LIN {X 0,Y 488.725,Z 497.921,A -85,B 0,C 180,E1 -6513.485,E2 -6513.485} C_VEL
LIN {X 0,Y 488.681,Z 497.925,A -85,B 0,C 180,E1 -6516.357,E2 -6516.357} C_VEL
LIN {X 0,Y 488.74,Z 497.918,A -85,B 0,C 180,E1 -6519.25,E2 -6519.25} C_VEL
LIN {X 0,Y 488.724,Z 497.922,A -85,B 0,C 180,E1 -6522.522,E2 -6522.522} C_VEL
LIN {X 0,Y 488.717,Z 498.007,A -85,B 0,C 180,E1 -6523.954,E2 -6523.954} C_VEL
LIN {X 0,Y 490.803,Z 507.385,A -85,B 0,C 180,E1 -6526.91,E2 -6526.91} C_VEL
LIN {X 0,Y 492.374,Z 514.903,A -85,B 0,C 180,E1 -6529.157,E2 -6529.157} C_VEL
LIN {X 0,Y 492.613,Z 519.318,A -85,B 0,C 180,E1 -6530.39,E2 -6530.39} C_VEL
LIN {X 0,Y 492.156,Z 529.697,A -85,B 0,C 180,E1 -6533.149,E2 -6533.149} C_VEL
LIN {X 0,Y 491.624,Z 540.769,A -85,B 0,C 180,E1 -6536.01,E2 -6536.01} C_VEL
LIN {X 0,Y 491.178,Z 552.868,A -85,B 0,C 180,E1 -6538.997,E2 -6538.997} C_VEL
LIN {X 0,Y 490.723,Z 566.378,A -85,B 0,C 180,E1 -6542.262,E2 -6542.262} C_VEL
LIN {X 0,Y 490.185,Z 577.141,A -85,B 0,C 180,E1 -6544.944,E2 -6544.944} C_VEL
LIN {X 0,Y 496.327,Z 599.12,A -85,B 0,C 180,E1 -6545.676,E2 -6545.676} C_VEL
LIN {X 0,Y 496.647,Z 602.392,A -85,B 0,C 180,E1 -6545.773,E2 -6545.773} C_VEL
LIN {X 0,Y 496.101,Z 618.413,A -85,B 0,C 180,E1 -6546.242,E2 -6546.242} C_VEL
LIN {X 0,Y 495.355,Z 634.974,A -85,B 0,C 180,E1 -6546.898,E2 -6546.898} C_VEL
LIN {X 0,Y 494.605,Z 650.253,A -85,B 0,C 180,E1 -6547.677,E2 -6547.677} C_VEL
LIN {X 0,Y 493.629,Z 665.049,A -85,B 0,C 180,E1 -6548.604,E2 -6548.604} C_VEL
LIN {X 0,Y 492.776,Z 678.915,A -85,B 0,C 180,E1 -6549.658,E2 -6549.658} C_VEL
LIN {X 0,Y 491.84,Z 691.852,A -85,B 0,C 180,E1 -6550.814,E2 -6550.814} C_VEL
LIN {X 0,Y 491.019,Z 703.949,A -85,B 0,C 180,E1 -6552.079,E2 -6552.079} C_VEL
LIN {X 0,Y 490.241,Z 715.847,A -85,B 0,C 180,E1 -6553.548,E2 -6553.548} C_VEL
LIN {X 0,Y 489.589,Z 726.058,A -85,B 0,C 180,E1 -6555.027,E2 -6555.027} C_VEL
LIN {X 0,Y 488.981,Z 735.94,A -85,B 0,C 180,E1 -6556.706,E2 -6556.706} C_VEL
LIN {X 0,Y 488.619,Z 744.242,A -85,B 0,C 180,E1 -6558.384,E2 -6558.384} C_VEL
LIN {X 0,Y 488.232,Z 751.104,A -85,B 0,C 180,E1 -6560.054,E2 -6560.054} C_VEL
LIN {X 0,Y 488.096,Z 756.719,A -85,B 0,C 180,E1 -6561.722,E2 -6561.722} C_VEL
LIN {X 0,Y 488.006,Z 761.657,A -85,B 0,C 180,E1 -6563.563,E2 -6563.563} C_VEL
LIN {X 0,Y 487.908,Z 764.636,A -85,B 0,C 180,E1 -6565.043,E2 -6565.043} C_VEL
LIN {X 0,Y 487.944,Z 767.091,A -85,B 0,C 180,E1 -6566.698,E2 -6566.698} C_VEL
LIN {X 0,Y 487.884,Z 768.479,A -85,B 0,C 180,E1 -6568.35,E2 -6568.35} C_VEL
LIN {X 0,Y 487.814,Z 769,A -85,B 0,C 180,E1 -6570.001,E2 -6570.001} C_VEL
LIN {X 0,Y 487.884,Z 768.478,A -85,B 0,C 180,E1 -6571.652,E2 -6571.652} C_VEL
LIN {X 0,Y 487.944,Z 767.088,A -85,B 0,C 180,E1 -6573.304,E2 -6573.304} C_VEL
LIN {X 0,Y 487.909,Z 764.633,A -85,B 0,C 180,E1 -6574.959,E2 -6574.959} C_VEL
LIN {X 0,Y 488.028,Z 761.249,A -85,B 0,C 180,E1 -6576.616,E2 -6576.616} C_VEL
LIN {X 0,Y 488.124,Z 755.465,A -85,B 0,C 180,E1 -6578.696,E2 -6578.696} C_VEL
LIN {X 0,Y 488.432,Z 747.853,A -85,B 0,C 180,E1 -6580.782,E2 -6580.782} C_VEL
LIN {X 0,Y 488.824,Z 739.251,A -85,B 0,C 180,E1 -6582.666,E2 -6582.666} C_VEL
LIN {X 0,Y 489.347,Z 729.973,A -85,B 0,C 180,E1 -6584.345,E2 -6584.345} C_VEL
LIN {X 0,Y 489.928,Z 720.416,A -85,B 0,C 180,E1 -6585.817,E2 -6585.817} C_VEL
LIN {X 0,Y 490.659,Z 709.277,A -85,B 0,C 180,E1 -6587.291,E2 -6587.291} C_VEL
LIN {X 0,Y 491.496,Z 697.133,A -85,B 0,C 180,E1 -6588.66,E2 -6588.66} C_VEL
LIN {X 0,Y 492.417,Z 683.772,A -85,B 0,C 180,E1 -6589.932,E2 -6589.932} C_VEL
LIN {X 0,Y 493.382,Z 669.408,A -85,B 0,C 180,E1 -6591.081,E2 -6591.081} C_VEL
LIN {X 0,Y 494.346,Z 654.423,A -85,B 0,C 180,E1 -6592.075,E2 -6592.075} C_VEL
LIN {X 0,Y 495.141,Z 640.233,A -85,B 0,C 180,E1 -6592.854,E2 -6592.854} C_VEL
LIN {X 0,Y 495.855,Z 625.368,A -85,B 0,C 180,E1 -6593.504,E2 -6593.504} C_VEL
LIN {X 0,Y 496.412,Z 608.983,A -85,B 0,C 180,E1 -6594.055,E2 -6594.055} C_VEL
LIN {X 0,Y 496.555,Z 600.107,A -85,B 0,C 180,E1 -6594.288,E2 -6594.288} C_VEL
LIN {X 0,Y 490.963,Z 580.048,A -85,B 0,C 180,E1 -6594.966,E2 -6594.966} C_VEL
LIN {X 0,Y 490.197,Z 577.068,A -85,B 0,C 180,E1 -6595.073,E2 -6595.073} C_VEL
LIN {X 0,Y 490.764,Z 564.422,A -85,B 0,C 180,E1 -6598.202,E2 -6598.202} C_VEL
LIN {X 0,Y 491.068,Z 550.504,A -85,B 0,C 180,E1 -6601.252,E2 -6601.252} C_VEL
LIN {X 0,Y 491.235,Z 537.358,A -85,B 0,C 180,E1 -6604.163,E2 -6604.163} C_VEL
LIN {X 0,Y 491.399,Z 525.732,A -85,B 0,C 180,E1 -6606.783,E2 -6606.783} C_VEL
LIN {X 0,Y 491.485,Z 513.366,A -85,B 0,C 180,E1 -6609.707,E2 -6609.707} C_VEL
LIN {X 0,Y 490.808,Z 508.373,A -85,B 0,C 180,E1 -6611,E2 -6611} C_VEL
LIN {X 0,Y 489.018,Z 499.36,A -85,B 0,C 180,E1 -6613.618,E2 -6613.618} C_VEL
LIN {X 0,Y 488.71,Z 497.924,A -85,B 0,C 180,E1 -6614.132,E2 -6614.132} C_VEL
LIN {X 0,Y 488.716,Z 497.923,A -85,B 0,C 180,E1 -6617.173,E2 -6617.173} C_VEL
LIN {X 0,Y 488.734,Z 497.919,A -85,B 0,C 180,E1 -6619.677,E2 -6619.677} C_VEL
LIN {X 0,Y 488.683,Z 497.927,A -85,B 0,C 180,E1 -6622.842,E2 -6622.842} C_VEL
LIN {X 0,Y 488.735,Z 497.92,A -85,B 0,C 180,E1 -6625.888,E2 -6625.888} C_VEL
LIN {X 0,Y 488.694,Z 497.925,A -85,B 0,C 180,E1 -6628.821,E2 -6628.821} C_VEL
LIN {X 0,Y 488.747,Z 497.919,A -85,B 0,C 180,E1 -6631.672,E2 -6631.672} C_VEL
LIN {X 0,Y 488.749,Z 497.919,A -85,B 0,C 180,E1 -6634.445,E2 -6634.445} C_VEL
LIN {X 0,Y 488.776,Z 498.087,A -85,B 0,C 180,E1 -6635.425,E2 -6635.425} C_VEL
LIN {X 0,Y 491.571,Z 505.225,A -85,B 0,C 180,E1 -6635.733,E2 -6635.733} C_VEL
LIN {X 0,Y 495.968,Z 516.083,A -85,B 0,C 180,E1 -6636.261,E2 -6636.261} C_VEL
LIN {X 0,Y 495.474,Z 531.577,A -85,B 0,C 180,E1 -6636.821,E2 -6636.821} C_VEL
LIN {X 0,Y 494.777,Z 546.893,A -85,B 0,C 180,E1 -6637.528,E2 -6637.528} C_VEL
LIN {X 0,Y 493.954,Z 562.027,A -85,B 0,C 180,E1 -6638.399,E2 -6638.399} C_VEL
LIN {X 0,Y 493.106,Z 576.875,A -85,B 0,C 180,E1 -6639.454,E2 -6639.454} C_VEL
LIN {X 0,Y 492.154,Z 590.761,A -85,B 0,C 180,E1 -6640.643,E2 -6640.643} C_VEL
LIN {X 0,Y 491.351,Z 602.834,A -85,B 0,C 180,E1 -6641.875,E2 -6641.875} C_VEL
LIN {X 0,Y 490.498,Z 615.066,A -85,B 0,C 180,E1 -6643.348,E2 -6643.348} C_VEL
LIN {X 0,Y 489.846,Z 625.403,A -85,B 0,C 180,E1 -6644.821,E2 -6644.821} C_VEL
LIN {X 0,Y 489.215,Z 634.165,A -85,B 0,C 180,E1 -6646.289,E2 -6646.289} C_VEL
LIN {X 0,Y 488.786,Z 643.123,A -85,B 0,C 180,E1 -6648.079,E2 -6648.079} C_VEL
LIN {X 0,Y 488.353,Z 649.619,A -85,B 0,C 180,E1 -6649.637,E2 -6649.637} C_VEL
LIN {X 0,Y 488.136,Z 655.35,A -85,B 0,C 180,E1 -6651.305,E2 -6651.305} C_VEL
LIN {X 0,Y 488.047,Z 660.122,A -85,B 0,C 180,E1 -6652.97,E2 -6652.97} C_VEL
LIN {X 0,Y 487.91,Z 664.571,A -85,B 0,C 180,E1 -6655.042,E2 -6655.042} C_VEL
LIN {X 0,Y 487.947,Z 667.016,A -85,B 0,C 180,E1 -6656.698,E2 -6656.698} C_VEL
LIN {X 0,Y 487.884,Z 668.488,A -85,B 0,C 180,E1 -6658.349,E2 -6658.349} C_VEL
LIN {X 0,Y 487.817,Z 668.997,A -85,B 0,C 180,E1 -6660,E2 -6660} C_VEL
LIN {X 0,Y 487.884,Z 668.527,A -85,B 0,C 180,E1 -6661.651,E2 -6661.651} C_VEL
LIN {X 0,Y 487.948,Z 667.112,A -85,B 0,C 180,E1 -6663.303,E2 -6663.303} C_VEL
LIN {X 0,Y 487.91,Z 664.728,A -85,B 0,C 180,E1 -6664.958,E2 -6664.958} C_VEL
LIN {X 0,Y 488.032,Z 661.294,A -85,B 0,C 180,E1 -6666.633,E2 -6666.633} C_VEL
LIN {X 0,Y 488.096,Z 656.884,A -85,B 0,C 180,E1 -6668.279,E2 -6668.279} C_VEL
LIN {X 0,Y 488.339,Z 649.846,A -85,B 0,C 180,E1 -6670.364,E2 -6670.364} C_VEL
LIN {X 0,Y 488.751,Z 642.59,A -85,B 0,C 180,E1 -6672.093,E2 -6672.093} C_VEL
LIN {X 0,Y 489.171,Z 634.413,A -85,B 0,C 180,E1 -6673.713,E2 -6673.713} C_VEL
LIN {X 0,Y 489.861,Z 624.292,A -85,B 0,C 180,E1 -6675.392,E2 -6675.392} C_VEL
LIN {X 0,Y 490.52,Z 613.752,A -85,B 0,C 180,E1 -6676.866,E2 -6676.866} C_VEL
LIN {X 0,Y 491.346,Z 601.265,A -85,B 0,C 180,E1 -6678.342,E2 -6678.342} C_VEL
LIN {X 0,Y 492.299,Z 588.147,A -85,B 0,C 180,E1 -6679.646,E2 -6679.646} C_VEL
LIN {X 0,Y 493.142,Z 574.876,A -85,B 0,C 180,E1 -6680.764,E2 -6680.764} C_VEL
LIN {X 0,Y 494.088,Z 560.086,A -85,B 0,C 180,E1 -6681.8,E2 -6681.8} C_VEL
LIN {X 0,Y 494.967,Z 543.931,A -85,B 0,C 180,E1 -6682.722,E2 -6682.722} C_VEL
LIN {X 0,Y 495.702,Z 527.836,A -85,B 0,C 180,E1 -6683.442,E2 -6683.442} C_VEL
LIN {X 0,Y 495.996,Z 515.787,A -85,B 0,C 180,E1 -6683.882,E2 -6683.882} C_VEL
LIN {X 0,Y 488.905,Z 498.693,A -85,B 0,C 180,E1 -6684.723,E2 -6684.723} C_VEL
LIN {X 0,Y 488.751,Z 497.919,A -85,B 0,C 180,E1 -6684.776,E2 -6684.776} C_VEL
LIN {X 0,Y 488.75,Z 497.919,A -85,B 0,C 180,E1 -6687.397,E2 -6687.397} C_VEL
LIN {X 0,Y 488.714,Z 497.924,A -85,B 0,C 180,E1 -6690.363,E2 -6690.363} C_VEL
LIN {X 0,Y 488.74,Z 497.92,A -85,B 0,C 180,E1 -6693.484,E2 -6693.484} C_VEL
LIN {X 0,Y 488.693,Z 497.925,A -85,B 0,C 180,E1 -6696.356,E2 -6696.356} C_VEL
LIN {X 0,Y 488.706,Z 497.923,A -85,B 0,C 180,E1 -6699.254,E2 -6699.254} C_VEL
LIN {X 0,Y 488.711,Z 497.924,A -85,B 0,C 180,E1 -6701.6,E2 -6701.6} C_VEL
LIN {X 0,Y 488.706,Z 497.924,A -85,B 0,C 180,E1 -6704.803,E2 -6704.803} C_VEL
LIN {X 0,Y 488.697,Z 497.927,A -85,B 0,C 180,E1 -6707.475,E2 -6707.475} C_VEL
LIN {X 0,Y 488.738,Z 497.918,A -85,B 0,C 180,E1 -6709.677,E2 -6709.677} C_VEL
LIN {X 0,Y 488.685,Z 497.926,A -85,B 0,C 180,E1 -6712.841,E2 -6712.841} C_VEL
LIN {X 0,Y 488.72,Z 497.921,A -85,B 0,C 180,E1 -6715.293,E2 -6715.293} C_VEL
LIN {X 0,Y 488.045,Z 498.009,A -85,B 0,C 180,E1 -6715.981,E2 -6715.981} C_VEL
LIN {X 0,Y 485.167,Z 498.367,A -85,B 0,C 180,E1 -6717.098,E2 -6717.098} C_VEL
LIN {X 0,Y 482.742,Z 498.669,A -85,B 0,C 180,E1 -6717.998,E2 -6717.998} C_VEL
LIN {X 0,Y 481.713,Z 498.799,A -85,B 0,C 180,E1 -6718.694,E2 -6718.694} C_VEL
LIN {X 0,Y 481.635,Z 498.805,A -85,B 0,C 180,E1 -6718.93,E2 -6718.93} C_VEL
LIN {X 0,Y 481.705,Z 498.797,A -85,B 0,C 180,E1 -6721.218,E2 -6721.218} C_VEL
LIN {X 0,Y 481.721,Z 498.795,A -85,B 0,C 180,E1 -6724.043,E2 -6724.043} C_VEL
LIN {X 0,Y 481.809,Z 498.814,A -85,B 0,C 180,E1 -6725.09,E2 -6725.09} C_VEL
LIN {X 0,Y 481.825,Z 503.568,A -85,B 0,C 180,E1 -6727.713,E2 -6727.713} C_VEL
LIN {X 0,Y 481.792,Z 508.356,A -85,B 0,C 180,E1 -6730.396,E2 -6730.396} C_VEL
LIN {X 0,Y 481.714,Z 512.928,A -85,B 0,C 180,E1 -6733.034,E2 -6733.034} C_VEL
LIN {X 0,Y 481.656,Z 517.34,A -85,B 0,C 180,E1 -6735.637,E2 -6735.637} C_VEL
LIN {X 0,Y 481.655,Z 521.628,A -85,B 0,C 180,E1 -6738.212,E2 -6738.212} C_VEL
LIN {X 0,Y 481.521,Z 523.894,A -85,B 0,C 180,E1 -6739.585,E2 -6739.585} C_VEL
LIN {X 0,Y 483.194,Z 528.751,A -85,B 0,C 180,E1 -6739.766,E2 -6739.766} C_VEL
LIN {X 0,Y 487.776,Z 541.51,A -85,B 0,C 180,E1 -6740.284,E2 -6740.284} C_VEL
LIN {X 0,Y 490.122,Z 549.845,A -85,B 0,C 180,E1 -6740.638,E2 -6740.638} C_VEL
LIN {X 0,Y 489.482,Z 566.262,A -85,B 0,C 180,E1 -6741.187,E2 -6741.187} C_VEL
LIN {X 0,Y 488.681,Z 581.972,A -85,B 0,C 180,E1 -6741.887,E2 -6741.887} C_VEL
LIN {X 0,Y 487.896,Z 595.778,A -85,B 0,C 180,E1 -6742.654,E2 -6742.654} C_VEL
LIN {X 0,Y 486.995,Z 609.618,A -85,B 0,C 180,E1 -6743.578,E2 -6743.578} C_VEL
LIN {X 0,Y 485.954,Z 623.681,A -85,B 0,C 180,E1 -6744.709,E2 -6744.709} C_VEL
LIN {X 0,Y 484.982,Z 636.591,A -85,B 0,C 180,E1 -6745.948,E2 -6745.948} C_VEL
LIN {X 0,Y 484.042,Z 648.549,A -85,B 0,C 180,E1 -6747.294,E2 -6747.294} C_VEL
LIN {X 0,Y 483.242,Z 659.576,A -85,B 0,C 180,E1 -6748.749,E2 -6748.749} C_VEL
LIN {X 0,Y 482.389,Z 670.303,A -85,B 0,C 180,E1 -6750.416,E2 -6750.416} C_VEL
LIN {X 0,Y 481.88,Z 679.281,A -85,B 0,C 180,E1 -6752.089,E2 -6752.089} C_VEL
LIN {X 0,Y 481.43,Z 686.808,A -85,B 0,C 180,E1 -6753.766,E2 -6753.766} C_VEL
LIN {X 0,Y 481.158,Z 693.144,A -85,B 0,C 180,E1 -6755.447,E2 -6755.447} C_VEL
LIN {X 0,Y 480.967,Z 699.432,A -85,B 0,C 180,E1 -6757.556,E2 -6757.556} C_VEL
LIN {X 0,Y 480.779,Z 703.245,A -85,B 0,C 180,E1 -6759.252,E2 -6759.252} C_VEL
LIN {X 0,Y 480.778,Z 706.068,A -85,B 0,C 180,E1 -6760.954,E2 -6760.954} C_VEL
LIN {X 0,Y 480.792,Z 707.203,A -85,B 0,C 180,E1 -6761.808,E2 -6761.808} C_VEL
LIN {X 0,Y 480.678,Z 708.608,A -85,B 0,C 180,E1 -6763.528,E2 -6763.528} C_VEL
LIN {X 0,Y 480.686,Z 708.958,A -85,B 0,C 180,E1 -6765.257,E2 -6765.257} C_VEL
LIN {X 0,Y 480.664,Z 708.286,A -85,B 0,C 180,E1 -6767.002,E2 -6767.002} C_VEL
LIN {X 0,Y 480.708,Z 707.376,A -85,B 0,C 180,E1 -6768.137,E2 -6768.137} C_VEL
LIN {X 0,Y 480.706,Z 705.387,A -85,B 0,C 180,E1 -6769.648,E2 -6769.648} C_VEL
LIN {X 0,Y 480.85,Z 702.058,A -85,B 0,C 180,E1 -6771.431,E2 -6771.431} C_VEL
LIN {X 0,Y 480.972,Z 697.519,A -85,B 0,C 180,E1 -6773.235,E2 -6773.235} C_VEL
LIN {X 0,Y 481.173,Z 693.316,A -85,B 0,C 180,E1 -6774.598,E2 -6774.598} C_VEL
LIN {X 0,Y 481.49,Z 686.376,A -85,B 0,C 180,E1 -6776.434,E2 -6776.434} C_VEL
LIN {X 0,Y 481.874,Z 679.039,A -85,B 0,C 180,E1 -6778.056,E2 -6778.056} C_VEL
LIN {X 0,Y 482.471,Z 670.265,A -85,B 0,C 180,E1 -6779.686,E2 -6779.686} C_VEL
LIN {X 0,Y 483.229,Z 659.526,A -85,B 0,C 180,E1 -6781.359,E2 -6781.359} C_VEL
LIN {X 0,Y 484.128,Z 648.196,A -85,B 0,C 180,E1 -6782.847,E2 -6782.847} C_VEL
LIN {X 0,Y 485.03,Z 636.036,A -85,B 0,C 180,E1 -6784.209,E2 -6784.209} C_VEL
LIN {X 0,Y 485.99,Z 623.103,A -85,B 0,C 180,E1 -6785.441,E2 -6785.441} C_VEL
LIN {X 0,Y 486.981,Z 609.495,A -85,B 0,C 180,E1 -6786.533,E2 -6786.533} C_VEL
LIN {X 0,Y 488.011,Z 593.857,A -85,B 0,C 180,E1 -6787.565,E2 -6787.565} C_VEL
LIN {X 0,Y 488.853,Z 578.577,A -85,B 0,C 180,E1 -6788.378,E2 -6788.378} C_VEL
LIN {X 0,Y 489.58,Z 563.019,A -85,B 0,C 180,E1 -6789.03,E2 -6789.03} C_VEL
LIN {X 0,Y 490.006,Z 549.235,A -85,B 0,C 180,E1 -6789.482,E2 -6789.482} C_VEL
LIN {X 0,Y 485.726,Z 535.434,A -85,B 0,C 180,E1 -6790.056,E2 -6790.056} C_VEL
LIN {X 0,Y 481.567,Z 524.772,A -85,B 0,C 180,E1 -6790.484,E2 -6790.484} C_VEL
LIN {X 0,Y 481.449,Z 524.174,A -85,B 0,C 180,E1 -6790.505,E2 -6790.505} C_VEL
LIN {X 0,Y 481.573,Z 519.519,A -85,B 0,C 180,E1 -6793.305,E2 -6793.305} C_VEL
LIN {X 0,Y 481.703,Z 515.606,A -85,B 0,C 180,E1 -6795.633,E2 -6795.633} C_VEL
LIN {X 0,Y 481.784,Z 509.992,A -85,B 0,C 180,E1 -6798.971,E2 -6798.971} C_VEL
LIN {X 0,Y 481.814,Z 504.644,A -85,B 0,C 180,E1 -6801.966,E2 -6801.966} C_VEL
LIN {X 0,Y 481.871,Z 500.416,A -85,B 0,C 180,E1 -6804.31,E2 -6804.31} C_VEL
LIN {X 0,Y 481.719,Z 498.796,A -85,B 0,C 180,E1 -6805.25,E2 -6805.25} C_VEL
LIN {X 0,Y 481.641,Z 498.808,A -85,B 0,C 180,E1 -6808.311,E2 -6808.311} C_VEL
LIN {X 0,Y 481.699,Z 498.797,A -85,B 0,C 180,E1 -6811.218,E2 -6811.218} C_VEL
LIN {X 0,Y 481.699,Z 498.797,A -85,B 0,C 180,E1 -6814.042,E2 -6814.042} C_VEL
LIN {X 0,Y 481.665,Z 498.799,A -85,B 0,C 180,E1 -6816.811,E2 -6816.811} C_VEL
LIN {X 0,Y 481.689,Z 498.798,A -85,B 0,C 180,E1 -6819.502,E2 -6819.502} C_VEL
LIN {X 0,Y 481.698,Z 498.797,A -85,B 0,C 180,E1 -6822.158,E2 -6822.158} C_VEL
LIN {X 0,Y 481.732,Z 498.792,A -85,B 0,C 180,E1 -6824.775,E2 -6824.775} C_VEL
LIN {X 0,Y 481.785,Z 498.787,A -85,B 0,C 180,E1 -6828.216,E2 -6828.216} C_VEL
LIN {X 0,Y 481.754,Z 498.785,A -85,B 0,C 180,E1 -6831.611,E2 -6831.611} C_VEL
LIN {X 0,Y 481.822,Z 498.78,A -85,B 0,C 180,E1 -6834.139,E2 -6834.139} C_VEL
LIN {X 0,Y 481.92,Z 498.768,A -85,B 0,C 180,E1 -6837.492,E2 -6837.492} C_VEL
LIN {X 0,Y 481.929,Z 498.767,A -85,B 0,C 180,E1 -6840,E2 -6840} C_VEL
LIN {X 0,Y 481.92,Z 498.766,A -85,B 0,C 180,E1 -6842.507,E2 -6842.507} C_VEL
LIN {X 0,Y 481.806,Z 498.777,A -85,B 0,C 180,E1 -6845.86,E2 -6845.86} C_VEL
LIN {X 0,Y 481.753,Z 498.786,A -85,B 0,C 180,E1 -6848.388,E2 -6848.388} C_VEL
LIN {X 0,Y 481.784,Z 498.781,A -85,B 0,C 180,E1 -6851.784,E2 -6851.784} C_VEL
LIN {X 0,Y 481.731,Z 498.79,A -85,B 0,C 180,E1 -6855.224,E2 -6855.224} C_VEL
LIN {X 0,Y 481.701,Z 498.782,A -85,B 0,C 180,E1 -6858.722,E2 -6858.722} C_VEL
LIN {X 0,Y 481.661,Z 498.801,A -85,B 0,C 180,E1 -6861.394,E2 -6861.394} C_VEL
LIN {X 0,Y 481.671,Z 498.78,A -85,B 0,C 180,E1 -6864.113,E2 -6864.113} C_VEL
LIN {X 0,Y 481.741,Z 498.79,A -85,B 0,C 180,E1 -6867.141,E2 -6867.141} C_VEL
LIN {X 0,Y 481.677,Z 498.798,A -85,B 0,C 180,E1 -6869.741,E2 -6869.741} C_VEL
LIN {X 0,Y 481.663,Z 498.8,A -85,B 0,C 180,E1 -6872.674,E2 -6872.674} C_VEL
LIN {X 0,Y 481.634,Z 498.803,A -85,B 0,C 180,E1 -6875.709,E2 -6875.709} C_VEL
LIN {X 0,Y 481.713,Z 498.793,A -85,B 0,C 180,E1 -6879.356,E2 -6879.356} C_VEL
LIN {X 0,Y 481.666,Z 498.801,A -85,B 0,C 180,E1 -6882.158,E2 -6882.158} C_VEL
LIN {X 0,Y 481.684,Z 498.854,A -85,B 0,C 180,E1 -6883.51,E2 -6883.51} C_VEL
LIN {X 0,Y 483.777,Z 508.43,A -85,B 0,C 180,E1 -6886.582,E2 -6886.582} C_VEL
LIN {X 0,Y 485.385,Z 515.824,A -85,B 0,C 180,E1 -6888.843,E2 -6888.843} C_VEL
LIN {X 0,Y 485.754,Z 520.091,A -85,B 0,C 180,E1 -6890.068,E2 -6890.068} C_VEL
LIN {X 0,Y 485.357,Z 529.232,A -85,B 0,C 180,E1 -6892.545,E2 -6892.545} C_VEL
LIN {X 0,Y 484.909,Z 538.824,A -85,B 0,C 180,E1 -6895.077,E2 -6895.077} C_VEL
LIN {X 0,Y 484.371,Z 550.439,A -85,B 0,C 180,E1 -6898.023,E2 -6898.023} C_VEL
LIN {X 0,Y 483.892,Z 562.462,A -85,B 0,C 180,E1 -6900.988,E2 -6900.988} C_VEL
LIN {X 0,Y 483.456,Z 573.592,A -85,B 0,C 180,E1 -6903.682,E2 -6903.682} C_VEL
LIN {X 0,Y 483.296,Z 577.121,A -85,B 0,C 180,E1 -6904.557,E2 -6904.557} C_VEL
LIN {X 0,Y 489.432,Z 599.121,A -85,B 0,C 180,E1 -6905.311,E2 -6905.311} C_VEL
LIN {X 0,Y 490.174,Z 602.392,A -85,B 0,C 180,E1 -6905.432,E2 -6905.432} C_VEL
LIN {X 0,Y 489.584,Z 618.966,A -85,B 0,C 180,E1 -6905.926,E2 -6905.926} C_VEL
LIN {X 0,Y 488.79,Z 635.537,A -85,B 0,C 180,E1 -6906.598,E2 -6906.598} C_VEL
LIN {X 0,Y 487.97,Z 650.948,A -85,B 0,C 180,E1 -6907.401,E2 -6907.401} C_VEL
LIN {X 0,Y 486.966,Z 665.051,A -85,B 0,C 180,E1 -6908.296,E2 -6908.296} C_VEL
LIN {X 0,Y 486.072,Z 678.913,A -85,B 0,C 180,E1 -6909.365,E2 -6909.365} C_VEL
LIN {X 0,Y 484.978,Z 692.92,A -85,B 0,C 180,E1 -6910.642,E2 -6910.642} C_VEL
LIN {X 0,Y 484.036,Z 705.732,A -85,B 0,C 180,E1 -6912.03,E2 -6912.03} C_VEL
LIN {X 0,Y 483.198,Z 717.701,A -85,B 0,C 180,E1 -6913.56,E2 -6913.56} C_VEL
LIN {X 0,Y 482.561,Z 727.411,A -85,B 0,C 180,E1 -6915.019,E2 -6915.019} C_VEL
LIN {X 0,Y 481.902,Z 737.055,A -85,B 0,C 180,E1 -6916.722,E2 -6916.722} C_VEL
LIN {X 0,Y 481.612,Z 744.243,A -85,B 0,C 180,E1 -6918.213,E2 -6918.213} C_VEL
LIN {X 0,Y 481.185,Z 751.103,A -85,B 0,C 180,E1 -6919.907,E2 -6919.907} C_VEL
LIN {X 0,Y 481.023,Z 756.719,A -85,B 0,C 180,E1 -6921.6,E2 -6921.6} C_VEL
LIN {X 0,Y 480.917,Z 761.897,A -85,B 0,C 180,E1 -6923.58,E2 -6923.58} C_VEL
LIN {X 0,Y 480.834,Z 764.636,A -85,B 0,C 180,E1 -6924.97,E2 -6924.97} C_VEL
LIN {X 0,Y 480.849,Z 767.091,A -85,B 0,C 180,E1 -6926.649,E2 -6926.649} C_VEL
LIN {X 0,Y 480.785,Z 768.479,A -85,B 0,C 180,E1 -6928.326,E2 -6928.326} C_VEL
LIN {X 0,Y 480.738,Z 769,A -85,B 0,C 180,E1 -6930.001,E2 -6930.001} C_VEL
LIN {X 0,Y 480.785,Z 768.478,A -85,B 0,C 180,E1 -6931.676,E2 -6931.676} C_VEL
LIN {X 0,Y 480.85,Z 767.088,A -85,B 0,C 180,E1 -6933.352,E2 -6933.352} C_VEL
LIN {X 0,Y 480.835,Z 764.633,A -85,B 0,C 180,E1 -6935.032,E2 -6935.032} C_VEL
LIN {X 0,Y 480.951,Z 761.249,A -85,B 0,C 180,E1 -6936.714,E2 -6936.714} C_VEL
LIN {X 0,Y 481.058,Z 755.465,A -85,B 0,C 180,E1 -6938.825,E2 -6938.825} C_VEL
LIN {X 0,Y 481.399,Z 747.853,A -85,B 0,C 180,E1 -6940.941,E2 -6940.941} C_VEL
LIN {X 0,Y 481.822,Z 739.252,A -85,B 0,C 180,E1 -6942.853,E2 -6942.853} C_VEL
LIN {X 0,Y 482.366,Z 729.973,A -85,B 0,C 180,E1 -6944.557,E2 -6944.557} C_VEL
LIN {X 0,Y 482.998,Z 720.416,A -85,B 0,C 180,E1 -6946.05,E2 -6946.05} C_VEL
LIN {X 0,Y 483.784,Z 709.277,A -85,B 0,C 180,E1 -6947.545,E2 -6947.545} C_VEL
LIN {X 0,Y 484.702,Z 697.132,A -85,B 0,C 180,E1 -6948.932,E2 -6948.932} C_VEL
LIN {X 0,Y 485.686,Z 683.868,A -85,B 0,C 180,E1 -6950.211,E2 -6950.211} C_VEL
LIN {X 0,Y 486.61,Z 670.833,A -85,B 0,C 180,E1 -6951.278,E2 -6951.278} C_VEL
LIN {X 0,Y 487.614,Z 656.231,A -85,B 0,C 180,E1 -6952.282,E2 -6952.282} C_VEL
LIN {X 0,Y 488.479,Z 642.089,A -85,B 0,C 180,E1 -6953.083,E2 -6953.083} C_VEL
LIN {X 0,Y 489.274,Z 626.871,A -85,B 0,C 180,E1 -6953.775,E2 -6953.775} C_VEL
LIN {X 0,Y 489.863,Z 611.154,A -85,B 0,C 180,E1 -6954.33,E2 -6954.33} C_VEL
LIN {X 0,Y 490.106,Z 601.692,A -85,B 0,C 180,E1 -6954.589,E2 -6954.589} C_VEL
LIN {X 0,Y 485.5,Z 584.865,A -85,B 0,C 180,E1 -6955.189,E2 -6955.189} C_VEL
LIN {X 0,Y 483.293,Z 577.11,A -85,B 0,C 180,E1 -6955.446,E2 -6955.446} C_VEL
LIN {X 0,Y 483.562,Z 569.778,A -85,B 0,C 180,E1 -6957.178,E2 -6957.178} C_VEL
LIN {X 0,Y 483.873,Z 556.679,A -85,B 0,C 180,E1 -6960.073,E2 -6960.073} C_VEL
LIN {X 0,Y 484.154,Z 543.502,A -85,B 0,C 180,E1 -6963.02,E2 -6963.02} C_VEL
LIN {X 0,Y 484.358,Z 530.237,A -85,B 0,C 180,E1 -6966.041,E2 -6966.041} C_VEL
LIN {X 0,Y 484.561,Z 517.337,A -85,B 0,C 180,E1 -6969.118,E2 -6969.118} C_VEL
LIN {X 0,Y 484.476,Z 513.014,A -85,B 0,C 180,E1 -6970.211,E2 -6970.211} C_VEL
LIN {X 0,Y 482.812,Z 504.327,A -85,B 0,C 180,E1 -6972.686,E2 -6972.686} C_VEL
LIN {X 0,Y 481.674,Z 498.801,A -85,B 0,C 180,E1 -6974.529,E2 -6974.529} C_VEL
LIN {X 0,Y 481.655,Z 498.801,A -85,B 0,C 180,E1 -6977.841,E2 -6977.841} C_VEL
LIN {X 0,Y 481.682,Z 498.8,A -85,B 0,C 180,E1 -6980.652,E2 -6980.652} C_VEL
LIN {X 0,Y 481.631,Z 498.804,A -85,B 0,C 180,E1 -6983.376,E2 -6983.376} C_VEL
LIN {X 0,Y 481.711,Z 498.797,A -85,B 0,C 180,E1 -6986.331,E2 -6986.331} C_VEL
LIN {X 0,Y 481.652,Z 498.801,A -85,B 0,C 180,E1 -6989.418,E2 -6989.418} C_VEL
LIN {X 0,Y 481.702,Z 498.798,A -85,B 0,C 180,E1 -6992.169,E2 -6992.169} C_VEL
LIN {X 0,Y 481.709,Z 498.795,A -85,B 0,C 180,E1 -6995.072,E2 -6995.072} C_VEL
LIN {X 0,Y 483.396,Z 503.34,A -85,B 0,C 180,E1 -6995.264,E2 -6995.264} C_VEL
LIN {X 0,Y 489.358,Z 518.074,A -85,B 0,C 180,E1 -6996,E2 -6996} C_VEL
LIN {X 0,Y 488.788,Z 534.305,A -85,B 0,C 180,E1 -6996.612,E2 -6996.612} C_VEL
LIN {X 0,Y 488.059,Z 549.801,A -85,B 0,C 180,E1 -6997.362,E2 -6997.362} C_VEL
LIN {X 0,Y 487.142,Z 565.421,A -85,B 0,C 180,E1 -6998.304,E2 -6998.304} C_VEL
LIN {X 0,Y 486.265,Z 579.876,A -85,B 0,C 180,E1 -6999.373,E2 -6999.373} C_VEL
LIN {X 0,Y 485.354,Z 593.159,A -85,B 0,C 180,E1 -7000.547,E2 -7000.547} C_VEL
LIN {X 0,Y 484.466,Z 605.303,A -85,B 0,C 180,E1 -7001.827,E2 -7001.827} C_VEL
LIN {X 0,Y 483.608,Z 616.721,A -85,B 0,C 180,E1 -7003.242,E2 -7003.242} C_VEL
LIN {X 0,Y 482.857,Z 627.435,A -85,B 0,C 180,E1 -7004.812,E2 -7004.812} C_VEL
LIN {X 0,Y 482.251,Z 636.083,A -85,B 0,C 180,E1 -7006.302,E2 -7006.302} C_VEL
LIN {X 0,Y 481.851,Z 644.171,A -85,B 0,C 180,E1 -7007.966,E2 -7007.966} C_VEL
LIN {X 0,Y 481.283,Z 651.958,A -85,B 0,C 180,E1 -7009.908,E2 -7009.908} C_VEL
LIN {X 0,Y 481.096,Z 657.405,A -85,B 0,C 180,E1 -7011.6,E2 -7011.6} C_VEL
LIN {X 0,Y 480.983,Z 662.242,A -85,B 0,C 180,E1 -7013.515,E2 -7013.515} C_VEL
LIN {X 0,Y 480.837,Z 665.027,A -85,B 0,C 180,E1 -7014.969,E2 -7014.969} C_VEL
LIN {X 0,Y 480.87,Z 667.348,A -85,B 0,C 180,E1 -7016.649,E2 -7016.649} C_VEL
LIN {X 0,Y 480.814,Z 668.745,A -85,B 0,C 180,E1 -7018.325,E2 -7018.325} C_VEL
LIN {X 0,Y 480.741,Z 669.232,A -85,B 0,C 180,E1 -7020,E2 -7020} C_VEL
LIN {X 0,Y 480.814,Z 668.771,A -85,B 0,C 180,E1 -7021.676,E2 -7021.676} C_VEL
LIN {X 0,Y 480.871,Z 667.399,A -85,B 0,C 180,E1 -7023.352,E2 -7023.352} C_VEL
LIN {X 0,Y 480.837,Z 665.106,A -85,B 0,C 180,E1 -7025.032,E2 -7025.032} C_VEL
LIN {X 0,Y 480.983,Z 661.823,A -85,B 0,C 180,E1 -7026.713,E2 -7026.713} C_VEL
LIN {X 0,Y 481.088,Z 657.497,A -85,B 0,C 180,E1 -7028.401,E2 -7028.401} C_VEL
LIN {X 0,Y 481.239,Z 652.047,A -85,B 0,C 180,E1 -7030.093,E2 -7030.093} C_VEL
LIN {X 0,Y 481.645,Z 645.342,A -85,B 0,C 180,E1 -7031.788,E2 -7031.788} C_VEL
LIN {X 0,Y 482.082,Z 637.214,A -85,B 0,C 180,E1 -7033.489,E2 -7033.489} C_VEL
LIN {X 0,Y 482.745,Z 627.46,A -85,B 0,C 180,E1 -7035.192,E2 -7035.192} C_VEL
LIN {X 0,Y 483.451,Z 617.438,A -85,B 0,C 180,E1 -7036.676,E2 -7036.676} C_VEL
LIN {X 0,Y 484.285,Z 605.455,A -85,B 0,C 180,E1 -7038.181,E2 -7038.181} C_VEL
LIN {X 0,Y 485.288,Z 592.297,A -85,B 0,C 180,E1 -7039.568,E2 -7039.568} C_VEL
LIN {X 0,Y 486.218,Z 579.089,A -85,B 0,C 180,E1 -7040.741,E2 -7040.741} C_VEL
LIN {X 0,Y 487.11,Z 564.777,A -85,B 0,C 180,E1 -7041.81,E2 -7041.81} C_VEL
LIN {X 0,Y 488.058,Z 549.128,A -85,B 0,C 180,E1 -7042.769,E2 -7042.769} C_VEL
LIN {X 0,Y 488.876,Z 534.058,A -85,B 0,C 180,E1 -7043.512,E2 -7043.512} C_VEL
LIN {X 0,Y 489.465,Z 518.375,A -85,B 0,C 180,E1 -7044.122,E2 -7044.122} C_VEL
LIN {X 0,Y 483.817,Z 504.249,A -85,B 0,C 180,E1 -7044.851,E2 -7044.851} C_VEL
LIN {X 0,Y 481.806,Z 499.34,A -85,B 0,C 180,E1 -7045.086,E2 -7045.086} C_VEL
LIN {X 0,Y 481.713,Z 498.796,A -85,B 0,C 180,E1 -7045.117,E2 -7045.117} C_VEL
LIN {X 0,Y 481.704,Z 498.793,A -85,B 0,C 180,E1 -7047.832,E2 -7047.832} C_VEL
LIN {X 0,Y 481.65,Z 498.803,A -85,B 0,C 180,E1 -7050.711,E2 -7050.711} C_VEL
LIN {X 0,Y 481.702,Z 498.795,A -85,B 0,C 180,E1 -7053.733,E2 -7053.733} C_VEL
LIN {X 0,Y 481.634,Z 498.803,A -85,B 0,C 180,E1 -7056.747,E2 -7056.747} C_VEL
LIN {X 0,Y 481.682,Z 498.798,A -85,B 0,C 180,E1 -7059.94,E2 -7059.94} C_VEL
LIN {X 0,Y 481.643,Z 498.804,A -85,B 0,C 180,E1 -7063.3,E2 -7063.3} C_VEL
LIN {X 0,Y 481.659,Z 498.8,A -85,B 0,C 180,E1 -7065.641,E2 -7065.641} C_VEL
LIN {X 0,Y 481.662,Z 498.803,A -85,B 0,C 180,E1 -7068.958,E2 -7068.958} C_VEL
LIN {X 0,Y 481.66,Z 498.802,A -85,B 0,C 180,E1 -7071.993,E2 -7071.993} C_VEL
LIN {X 0,Y 481.694,Z 498.796,A -85,B 0,C 180,E1 -7075.318,E2 -7075.318} C_VEL
LIN {X 0,Y 481.651,Z 498.805,A -85,B 0,C 180,E1 -7078.311,E2 -7078.311} C_VEL
LIN {X 0,Y 481.635,Z 498.805,A -85,B 0,C 180,E1 -7078.93,E2 -7078.93} C_VEL
LIN {X 0,Y 480.981,Z 498.888,A -85,B 0,C 180,E1 -7079.628,E2 -7079.628} C_VEL
LIN {X 0,Y 478.127,Z 499.243,A -85,B 0,C 180,E1 -7080.761,E2 -7080.761} C_VEL
LIN {X 0,Y 475.732,Z 499.542,A -85,B 0,C 180,E1 -7081.675,E2 -7081.675} C_VEL
LIN {X 0,Y 474.742,Z 499.663,A -85,B 0,C 180,E1 -7082.381,E2 -7082.381} C_VEL
LIN {X 0,Y 474.682,Z 499.671,A -85,B 0,C 180,E1 -7082.62,E2 -7082.62} C_VEL
LIN {X 0,Y 474.783,Z 499.847,A -85,B 0,C 180,E1 -7085.046,E2 -7085.046} C_VEL
LIN {X 0,Y 474.827,Z 504.068,A -85,B 0,C 180,E1 -7087.366,E2 -7087.366} C_VEL
LIN {X 0,Y 474.775,Z 508.906,A -85,B 0,C 180,E1 -7090.094,E2 -7090.094} C_VEL
LIN {X 0,Y 474.71,Z 513.554,A -85,B 0,C 180,E1 -7092.776,E2 -7092.776} C_VEL
LIN {X 0,Y 474.635,Z 518.029,A -85,B 0,C 180,E1 -7095.42,E2 -7095.42} C_VEL
LIN {X 0,Y 474.618,Z 522.393,A -85,B 0,C 180,E1 -7098.035,E2 -7098.035} C_VEL
LIN {X 0,Y 474.513,Z 524.312,A -85,B 0,C 180,E1 -7099.189,E2 -7099.189} C_VEL
LIN {X 0,Y 476.366,Z 529.517,A -85,B 0,C 180,E1 -7099.386,E2 -7099.386} C_VEL
LIN {X 0,Y 481.417,Z 543.355,A -85,B 0,C 180,E1 -7099.976,E2 -7099.976} C_VEL
LIN {X 0,Y 483.599,Z 551.749,A -85,B 0,C 180,E1 -7100.338,E2 -7100.338} C_VEL
LIN {X 0,Y 482.94,Z 567.839,A -85,B 0,C 180,E1 -7100.893,E2 -7100.893} C_VEL
LIN {X 0,Y 482.111,Z 583.579,A -85,B 0,C 180,E1 -7101.617,E2 -7101.617} C_VEL
LIN {X 0,Y 481.205,Z 597.977,A -85,B 0,C 180,E1 -7102.446,E2 -7102.446} C_VEL
LIN {X 0,Y 480.154,Z 612.832,A -85,B 0,C 180,E1 -7103.486,E2 -7103.486} C_VEL
LIN {X 0,Y 479.099,Z 626.496,A -85,B 0,C 180,E1 -7104.633,E2 -7104.633} C_VEL
LIN {X 0,Y 478.007,Z 640.08,A -85,B 0,C 180,E1 -7105.994,E2 -7105.994} C_VEL
LIN {X 0,Y 477.017,Z 652.416,A -85,B 0,C 180,E1 -7107.466,E2 -7107.466} C_VEL
LIN {X 0,Y 476.14,Z 662.9,A -85,B 0,C 180,E1 -7108.942,E2 -7108.942} C_VEL
LIN {X 0,Y 475.313,Z 673.137,A -85,B 0,C 180,E1 -7110.634,E2 -7110.634} C_VEL
LIN {X 0,Y 474.841,Z 680.803,A -85,B 0,C 180,E1 -7112.12,E2 -7112.12} C_VEL
LIN {X 0,Y 474.395,Z 688.173,A -85,B 0,C 180,E1 -7113.822,E2 -7113.822} C_VEL
LIN {X 0,Y 474.106,Z 694.316,A -85,B 0,C 180,E1 -7115.528,E2 -7115.528} C_VEL
LIN {X 0,Y 473.931,Z 699.374,A -85,B 0,C 180,E1 -7117.24,E2 -7117.24} C_VEL
LIN {X 0,Y 473.82,Z 702.43,A -85,B 0,C 180,E1 -7118.529,E2 -7118.529} C_VEL
LIN {X 0,Y 473.703,Z 705.617,A -85,B 0,C 180,E1 -7120.254,E2 -7120.254} C_VEL
LIN {X 0,Y 473.689,Z 707.815,A -85,B 0,C 180,E1 -7121.987,E2 -7121.987} C_VEL
LIN {X 0,Y 473.587,Z 709.062,A -85,B 0,C 180,E1 -7123.734,E2 -7123.734} C_VEL
LIN {X 0,Y 473.594,Z 709.271,A -85,B 0,C 180,E1 -7125.492,E2 -7125.492} C_VEL
LIN {X 0,Y 473.596,Z 708.521,A -85,B 0,C 180,E1 -7127.264,E2 -7127.264} C_VEL
LIN {X 0,Y 473.6,Z 706.707,A -85,B 0,C 180,E1 -7129.053,E2 -7129.053} C_VEL
LIN {X 0,Y 473.762,Z 703.873,A -85,B 0,C 180,E1 -7130.855,E2 -7130.855} C_VEL
LIN {X 0,Y 473.868,Z 699.82,A -85,B 0,C 180,E1 -7132.68,E2 -7132.68} C_VEL
LIN {X 0,Y 474.102,Z 694.474,A -85,B 0,C 180,E1 -7134.522,E2 -7134.522} C_VEL
LIN {X 0,Y 474.442,Z 687.746,A -85,B 0,C 180,E1 -7136.383,E2 -7136.383} C_VEL
LIN {X 0,Y 474.882,Z 680.713,A -85,B 0,C 180,E1 -7138.001,E2 -7138.001} C_VEL
LIN {X 0,Y 475.452,Z 672.221,A -85,B 0,C 180,E1 -7139.632,E2 -7139.632} C_VEL
LIN {X 0,Y 476.24,Z 661.852,A -85,B 0,C 180,E1 -7141.319,E2 -7141.319} C_VEL
LIN {X 0,Y 477.219,Z 650.164,A -85,B 0,C 180,E1 -7142.918,E2 -7142.918} C_VEL
LIN {X 0,Y 478.212,Z 637.753,A -85,B 0,C 180,E1 -7144.356,E2 -7144.356} C_VEL
LIN {X 0,Y 479.277,Z 624.512,A -85,B 0,C 180,E1 -7145.652,E2 -7145.652} C_VEL
LIN {X 0,Y 480.382,Z 609.758,A -85,B 0,C 180,E1 -7146.856,E2 -7146.856} C_VEL
LIN {X 0,Y 481.472,Z 594.028,A -85,B 0,C 180,E1 -7147.905,E2 -7147.905} C_VEL
LIN {X 0,Y 482.367,Z 578.679,A -85,B 0,C 180,E1 -7148.727,E2 -7148.727} C_VEL
LIN {X 0,Y 483.142,Z 563.159,A -85,B 0,C 180,E1 -7149.38,E2 -7149.38} C_VEL
LIN {X 0,Y 483.504,Z 550.766,A -85,B 0,C 180,E1 -7149.796,E2 -7149.796} C_VEL
LIN {X 0,Y 479.561,Z 537.998,A -85,B 0,C 180,E1 -7150.353,E2 -7150.353} C_VEL
LIN {X 0,Y 474.506,Z 524.921,A -85,B 0,C 180,E1 -7150.896,E2 -7150.896} C_VEL
LIN {X 0,Y 474.462,Z 524.557,A -85,B 0,C 180,E1 -7150.935,E2 -7150.935} C_VEL
LIN {X 0,Y 474.563,Z 520.36,A -85,B 0,C 180,E1 -7153.475,E2 -7153.475} C_VEL
LIN {X 0,Y 474.681,Z 515.273,A -85,B 0,C 180,E1 -7156.507,E2 -7156.507} C_VEL
LIN {X 0,Y 474.82,Z 510.421,A -85,B 0,C 180,E1 -7159.363,E2 -7159.363} C_VEL
LIN {X 0,Y 474.832,Z 504.676,A -85,B 0,C 180,E1 -7162.638,E2 -7162.638} C_VEL
LIN {X 0,Y 474.827,Z 500.844,A -85,B 0,C 180,E1 -7164.742,E2 -7164.742} C_VEL
LIN {X 0,Y 474.672,Z 499.674,A -85,B 0,C 180,E1 -7165.505,E2 -7165.505} C_VEL
LIN {X 0,Y 474.595,Z 499.685,A -85,B 0,C 180,E1 -7168.782,E2 -7168.782} C_VEL
LIN {X 0,Y 474.642,Z 499.676,A -85,B 0,C 180,E1 -7171.717,E2 -7171.717} C_VEL
LIN {X 0,Y 474.679,Z 499.672,A -85,B 0,C 180,E1 -7174.572,E2 -7174.572} C_VEL
LIN {X 0,Y 474.598,Z 499.681,A -85,B 0,C 180,E1 -7177.355,E2 -7177.355} C_VEL
LIN {X 0,Y 474.648,Z 499.677,A -85,B 0,C 180,E1 -7180.089,E2 -7180.089} C_VEL
LIN {X 0,Y 474.642,Z 499.677,A -85,B 0,C 180,E1 -7182.774,E2 -7182.774} C_VEL
LIN {X 0,Y 474.639,Z 499.676,A -85,B 0,C 180,E1 -7185.42,E2 -7185.42} C_VEL
LIN {X 0,Y 474.729,Z 499.665,A -85,B 0,C 180,E1 -7188.038,E2 -7188.038} C_VEL
LIN {X 0,Y 474.719,Z 499.662,A -85,B 0,C 180,E1 -7191.486,E2 -7191.486} C_VEL
LIN {X 0,Y 474.782,Z 499.658,A -85,B 0,C 180,E1 -7194.052,E2 -7194.052} C_VEL
LIN {X 0,Y 474.886,Z 499.644,A -85,B 0,C 180,E1 -7197.455,E2 -7197.455} C_VEL
LIN {X 0,Y 474.867,Z 499.646,A -85,B 0,C 180,E1 -7200.848,E2 -7200.848} C_VEL
LIN {X 0,Y 474.886,Z 499.642,A -85,B 0,C 180,E1 -7202.544,E2 -7202.544} C_VEL
LIN {X 0,Y 474.769,Z 499.654,A -85,B 0,C 180,E1 -7205.947,E2 -7205.947} C_VEL
LIN {X 0,Y 474.718,Z 499.663,A -85,B 0,C 180,E1 -7208.513,E2 -7208.513} C_VEL
LIN {X 0,Y 474.727,Z 499.659,A -85,B 0,C 180,E1 -7211.961,E2 -7211.961} C_VEL
LIN {X 0,Y 474.669,Z 499.664,A -85,B 0,C 180,E1 -7215.768,E2 -7215.768} C_VEL
LIN {X 0,Y 474.654,Z 499.664,A -85,B 0,C 180,E1 -7219.01,E2 -7219.01} C_VEL
LIN {X 0,Y 474.626,Z 499.676,A -85,B 0,C 180,E1 -7221.727,E2 -7221.727} C_VEL
LIN {X 0,Y 474.651,Z 499.652,A -85,B 0,C 180,E1 -7224.493,E2 -7224.493} C_VEL
LIN {X 0,Y 474.687,Z 499.668,A -85,B 0,C 180,E1 -7227.339,E2 -7227.339} C_VEL
LIN {X 0,Y 474.599,Z 499.681,A -85,B 0,C 180,E1 -7230.812,E2 -7230.812} C_VEL
LIN {X 0,Y 474.628,Z 499.675,A -85,B 0,C 180,E1 -7233.985,E2 -7233.985} C_VEL
LIN {X 0,Y 474.568,Z 499.682,A -85,B 0,C 180,E1 -7236.901,E2 -7236.901} C_VEL
LIN {X 0,Y 474.657,Z 499.672,A -85,B 0,C 180,E1 -7239.654,E2 -7239.654} C_VEL
LIN {X 0,Y 474.663,Z 499.792,A -85,B 0,C 180,E1 -7243.087,E2 -7243.087} C_VEL
LIN {X 0,Y 476.781,Z 509.467,A -85,B 0,C 180,E1 -7246.243,E2 -7246.243} C_VEL
LIN {X 0,Y 478.427,Z 517.093,A -85,B 0,C 180,E1 -7248.622,E2 -7248.622} C_VEL
LIN {X 0,Y 478.881,Z 521.025,A -85,B 0,C 180,E1 -7249.781,E2 -7249.781} C_VEL
LIN {X 0,Y 478.626,Z 527.227,A -85,B 0,C 180,E1 -7251.498,E2 -7251.498} C_VEL
LIN {X 0,Y 478.089,Z 538.369,A -85,B 0,C 180,E1 -7254.505,E2 -7254.505} C_VEL
LIN {X 0,Y 477.505,Z 549.948,A -85,B 0,C 180,E1 -7257.507,E2 -7257.507} C_VEL
LIN {X 0,Y 476.927,Z 563.508,A -85,B 0,C 180,E1 -7260.905,E2 -7260.905} C_VEL
LIN {X 0,Y 476.42,Z 575.039,A -85,B 0,C 180,E1 -7263.735,E2 -7263.735} C_VEL
LIN {X 0,Y 476.356,Z 576.761,A -85,B 0,C 180,E1 -7264.154,E2 -7264.154} C_VEL
LIN {X 0,Y 482.61,Z 599.216,A -85,B 0,C 180,E1 -7264.941,E2 -7264.941} C_VEL
LIN {X 0,Y 483.698,Z 603.599,A -85,B 0,C 180,E1 -7265.111,E2 -7265.111} C_VEL
LIN {X 0,Y 483.042,Z 620.062,A -85,B 0,C 180,E1 -7265.62,E2 -7265.62} C_VEL
LIN {X 0,Y 482.194,Z 636.665,A -85,B 0,C 180,E1 -7266.315,E2 -7266.315} C_VEL
LIN {X 0,Y 481.228,Z 652.591,A -85,B 0,C 180,E1 -7267.172,E2 -7267.172} C_VEL
LIN {X 0,Y 480.224,Z 666.579,A -85,B 0,C 180,E1 -7268.089,E2 -7268.089} C_VEL
LIN {X 0,Y 479.168,Z 681.488,A -85,B 0,C 180,E1 -7269.279,E2 -7269.279} C_VEL
LIN {X 0,Y 478.061,Z 695.055,A -85,B 0,C 180,E1 -7270.574,E2 -7270.574} C_VEL
LIN {X 0,Y 477.073,Z 707.512,A -85,B 0,C 180,E1 -7271.98,E2 -7271.98} C_VEL
LIN {X 0,Y 476.193,Z 719.093,A -85,B 0,C 180,E1 -7273.518,E2 -7273.518} C_VEL
LIN {X 0,Y 475.517,Z 728.745,A -85,B 0,C 180,E1 -7275.011,E2 -7275.011} C_VEL
LIN {X 0,Y 474.859,Z 738.17,A -85,B 0,C 180,E1 -7276.739,E2 -7276.739} C_VEL
LIN {X 0,Y 474.452,Z 746.053,A -85,B 0,C 180,E1 -7278.466,E2 -7278.466} C_VEL
LIN {X 0,Y 474.072,Z 752.628,A -85,B 0,C 180,E1 -7280.185,E2 -7280.185} C_VEL
LIN {X 0,Y 473.922,Z 757.959,A -85,B 0,C 180,E1 -7281.902,E2 -7281.902} C_VEL
LIN {X 0,Y 473.838,Z 762.113,A -85,B 0,C 180,E1 -7283.588,E2 -7283.588} C_VEL
LIN {X 0,Y 473.762,Z 764.636,A -85,B 0,C 180,E1 -7284.895,E2 -7284.895} C_VEL
LIN {X 0,Y 473.743,Z 767.092,A -85,B 0,C 180,E1 -7286.599,E2 -7286.599} C_VEL
LIN {X 0,Y 473.69,Z 768.479,A -85,B 0,C 180,E1 -7288.301,E2 -7288.301} C_VEL
LIN {X 0,Y 473.665,Z 769,A -85,B 0,C 180,E1 -7290.001,E2 -7290.001} C_VEL
LIN {X 0,Y 473.69,Z 768.477,A -85,B 0,C 180,E1 -7291.701,E2 -7291.701} C_VEL
LIN {X 0,Y 473.743,Z 767.088,A -85,B 0,C 180,E1 -7293.403,E2 -7293.403} C_VEL
LIN {X 0,Y 473.763,Z 764.632,A -85,B 0,C 180,E1 -7295.107,E2 -7295.107} C_VEL
LIN {X 0,Y 473.883,Z 761.25,A -85,B 0,C 180,E1 -7296.815,E2 -7296.815} C_VEL
LIN {X 0,Y 474.007,Z 755.465,A -85,B 0,C 180,E1 -7298.957,E2 -7298.957} C_VEL
LIN {X 0,Y 474.352,Z 747.852,A -85,B 0,C 180,E1 -7301.106,E2 -7301.106} C_VEL
LIN {X 0,Y 474.749,Z 740.264,A -85,B 0,C 180,E1 -7302.83,E2 -7302.83} C_VEL
LIN {X 0,Y 475.334,Z 731.203,A -85,B 0,C 180,E1 -7304.558,E2 -7304.558} C_VEL
LIN {X 0,Y 475.992,Z 721.901,A -85,B 0,C 180,E1 -7306.073,E2 -7306.073} C_VEL
LIN {X 0,Y 476.806,Z 710.999,A -85,B 0,C 180,E1 -7307.588,E2 -7307.588} C_VEL
LIN {X 0,Y 477.658,Z 700.056,A -85,B 0,C 180,E1 -7308.887,E2 -7308.887} C_VEL
LIN {X 0,Y 478.707,Z 687.329,A -85,B 0,C 180,E1 -7310.187,E2 -7310.187} C_VEL
LIN {X 0,Y 479.748,Z 673.679,A -85,B 0,C 180,E1 -7311.371,E2 -7311.371} C_VEL
LIN {X 0,Y 480.813,Z 659.074,A -85,B 0,C 180,E1 -7312.423,E2 -7312.423} C_VEL
LIN {X 0,Y 481.622,Z 646.058,A -85,B 0,C 180,E1 -7313.204,E2 -7313.204} C_VEL
LIN {X 0,Y 482.546,Z 630.821,A -85,B 0,C 180,E1 -7313.953,E2 -7313.953} C_VEL
LIN {X 0,Y 483.364,Z 614.72,A -85,B 0,C 180,E1 -7314.563,E2 -7314.563} C_VEL
LIN {X 0,Y 483.559,Z 603.077,A -85,B 0,C 180,E1 -7314.91,E2 -7314.91} C_VEL
LIN {X 0,Y 479.647,Z 588.338,A -85,B 0,C 180,E1 -7315.451,E2 -7315.451} C_VEL
LIN {X 0,Y 476.382,Z 577.091,A -85,B 0,C 180,E1 -7315.824,E2 -7315.824} C_VEL
LIN {X 0,Y 476.325,Z 576.221,A -85,B 0,C 180,E1 -7315.876,E2 -7315.876} C_VEL
LIN {X 0,Y 476.705,Z 562.839,A -85,B 0,C 180,E1 -7318.871,E2 -7318.871} C_VEL
LIN {X 0,Y 477.022,Z 548.855,A -85,B 0,C 180,E1 -7322.032,E2 -7322.032} C_VEL
LIN {X 0,Y 477.345,Z 533.868,A -85,B 0,C 180,E1 -7325.487,E2 -7325.487} C_VEL
LIN {X 0,Y 477.53,Z 521.55,A -85,B 0,C 180,E1 -7328.461,E2 -7328.461} C_VEL
LIN {X 0,Y 477.588,Z 515.227,A -85,B 0,C 180,E1 -7330.075,E2 -7330.075} C_VEL
LIN {X 0,Y 476.136,Z 507.079,A -85,B 0,C 180,E1 -7332.437,E2 -7332.437} C_VEL
LIN {X 0,Y 474.757,Z 500.381,A -85,B 0,C 180,E1 -7334.72,E2 -7334.72} C_VEL
LIN {X 0,Y 474.641,Z 499.677,A -85,B 0,C 180,E1 -7335.039,E2 -7335.039} C_VEL
LIN {X 0,Y 474.63,Z 499.678,A -85,B 0,C 180,E1 -7338.216,E2 -7338.216} C_VEL
LIN {X 0,Y 474.646,Z 499.677,A -85,B 0,C 180,E1 -7340.455,E2 -7340.455} C_VEL
LIN {X 0,Y 474.593,Z 499.681,A -85,B 0,C 180,E1 -7343.677,E2 -7343.677} C_VEL
LIN {X 0,Y 474.644,Z 499.675,A -85,B 0,C 180,E1 -7346.78,E2 -7346.78} C_VEL
LIN {X 0,Y 474.606,Z 499.68,A -85,B 0,C 180,E1 -7349.77,E2 -7349.77} C_VEL
LIN {X 0,Y 474.699,Z 499.669,A -85,B 0,C 180,E1 -7352.68,E2 -7352.68} C_VEL
LIN {X 0,Y 474.674,Z 499.672,A -85,B 0,C 180,E1 -7354.687,E2 -7354.687} C_VEL
LIN {X 0,Y 476.378,Z 504.145,A -85,B 0,C 180,E1 -7354.9,E2 -7354.9} C_VEL
LIN {X 0,Y 482.79,Z 520.07,A -85,B 0,C 180,E1 -7355.731,E2 -7355.731} C_VEL
LIN {X 0,Y 482.183,Z 536.334,A -85,B 0,C 180,E1 -7356.365,E2 -7356.365} C_VEL
LIN {X 0,Y 481.389,Z 551.857,A -85,B 0,C 180,E1 -7357.141,E2 -7357.141} C_VEL
LIN {X 0,Y 480.459,Z 567.26,A -85,B 0,C 180,E1 -7358.099,E2 -7358.099} C_VEL
LIN {X 0,Y 479.539,Z 581.553,A -85,B 0,C 180,E1 -7359.182,E2 -7359.182} C_VEL
LIN {X 0,Y 478.591,Z 594.737,A -85,B 0,C 180,E1 -7360.372,E2 -7360.372} C_VEL
LIN {X 0,Y 477.592,Z 607.774,A -85,B 0,C 180,E1 -7361.778,E2 -7361.778} C_VEL
LIN {X 0,Y 476.649,Z 619.65,A -85,B 0,C 180,E1 -7363.308,E2 -7363.308} C_VEL
LIN {X 0,Y 475.928,Z 629.45,A -85,B 0,C 180,E1 -7364.805,E2 -7364.805} C_VEL
LIN {X 0,Y 475.211,Z 639.014,A -85,B 0,C 180,E1 -7366.531,E2 -7366.531} C_VEL
LIN {X 0,Y 474.831,Z 646.067,A -85,B 0,C 180,E1 -7368.041,E2 -7368.041} C_VEL
LIN {X 0,Y 474.322,Z 652.769,A -85,B 0,C 180,E1 -7369.759,E2 -7369.759} C_VEL
LIN {X 0,Y 474.105,Z 658.236,A -85,B 0,C 180,E1 -7371.476,E2 -7371.476} C_VEL
LIN {X 0,Y 473.98,Z 663.131,A -85,B 0,C 180,E1 -7373.441,E2 -7373.441} C_VEL
LIN {X 0,Y 473.825,Z 665.858,A -85,B 0,C 180,E1 -7374.895,E2 -7374.895} C_VEL
LIN {X 0,Y 473.828,Z 668.185,A -85,B 0,C 180,E1 -7376.599,E2 -7376.599} C_VEL
LIN {X 0,Y 473.761,Z 669.559,A -85,B 0,C 180,E1 -7378.3,E2 -7378.3} C_VEL
LIN {X 0,Y 473.687,Z 670.039,A -85,B 0,C 180,E1 -7380,E2 -7380} C_VEL
LIN {X 0,Y 473.759,Z 669.567,A -85,B 0,C 180,E1 -7381.701,E2 -7381.701} C_VEL
LIN {X 0,Y 473.828,Z 668.17,A -85,B 0,C 180,E1 -7383.402,E2 -7383.402} C_VEL
LIN {X 0,Y 473.804,Z 665.844,A -85,B 0,C 180,E1 -7385.106,E2 -7385.106} C_VEL
LIN {X 0,Y 473.987,Z 661.55,A -85,B 0,C 180,E1 -7387.241,E2 -7387.241} C_VEL
LIN {X 0,Y 474.115,Z 656.905,A -85,B 0,C 180,E1 -7388.955,E2 -7388.955} C_VEL
LIN {X 0,Y 474.356,Z 651.097,A -85,B 0,C 180,E1 -7390.673,E2 -7390.673} C_VEL
LIN {X 0,Y 474.842,Z 643.685,A -85,B 0,C 180,E1 -7392.467,E2 -7392.467} C_VEL
LIN {X 0,Y 475.335,Z 635.493,A -85,B 0,C 180,E1 -7394.121,E2 -7394.121} C_VEL
LIN {X 0,Y 476.119,Z 625.24,A -85,B 0,C 180,E1 -7395.848,E2 -7395.848} C_VEL
LIN {X 0,Y 476.852,Z 614.573,A -85,B 0,C 180,E1 -7397.365,E2 -7397.365} C_VEL
LIN {X 0,Y 477.665,Z 603.9,A -85,B 0,C 180,E1 -7398.664,E2 -7398.664} C_VEL
LIN {X 0,Y 478.672,Z 591.045,A -85,B 0,C 180,E1 -7400.004,E2 -7400.004} C_VEL
LIN {X 0,Y 479.73,Z 576.685,A -85,B 0,C 180,E1 -7401.259,E2 -7401.259} C_VEL
LIN {X 0,Y 480.777,Z 561.764,A -85,B 0,C 180,E1 -7402.338,E2 -7402.338} C_VEL
LIN {X 0,Y 481.62,Z 547.218,A -85,B 0,C 180,E1 -7403.204,E2 -7403.204} C_VEL
LIN {X 0,Y 482.472,Z 531.466,A -85,B 0,C 180,E1 -7403.957,E2 -7403.957} C_VEL
LIN {X 0,Y 482.834,Z 519.754,A -85,B 0,C 180,E1 -7404.418,E2 -7404.418} C_VEL
LIN {X 0,Y 476.593,Z 504.677,A -85,B 0,C 180,E1 -7405.232,E2 -7405.232} C_VEL
LIN {X 0,Y 474.777,Z 500.349,A -85,B 0,C 180,E1 -7405.448,E2 -7405.448} C_VEL
LIN {X 0,Y 474.67,Z 499.673,A -85,B 0,C 180,E1 -7405.476,E2 -7405.476} C_VEL
LIN {X 0,Y 474.65,Z 499.672,A -85,B 0,C 180,E1 -7408.283,E2 -7408.283} C_VEL
LIN {X 0,Y 474.603,Z 499.68,A -85,B 0,C 180,E1 -7411.218,E2 -7411.218} C_VEL
LIN {X 0,Y 474.638,Z 499.676,A -85,B 0,C 180,E1 -7414.241,E2 -7414.241} C_VEL
LIN {X 0,Y 474.597,Z 499.683,A -85,B 0,C 180,E1 -7417.384,E2 -7417.384} C_VEL
LIN {X 0,Y 474.632,Z 499.675,A -85,B 0,C 180,E1 -7419.648,E2 -7419.648} C_VEL
LIN {X 0,Y 474.619,Z 499.679,A -85,B 0,C 180,E1 -7422.934,E2 -7422.934} C_VEL
LIN {X 0,Y 474.611,Z 499.68,A -85,B 0,C 180,E1 -7425.895,E2 -7425.895} C_VEL
LIN {X 0,Y 474.634,Z 499.678,A -85,B 0,C 180,E1 -7429.041,E2 -7429.041} C_VEL
LIN {X 0,Y 474.615,Z 499.681,A -85,B 0,C 180,E1 -7431.704,E2 -7431.704} C_VEL
LIN {X 0,Y 474.63,Z 499.679,A -85,B 0,C 180,E1 -7434.726,E2 -7434.726} C_VEL
LIN {X 0,Y 474.641,Z 499.68,A -85,B 0,C 180,E1 -7437.788,E2 -7437.788} C_VEL
LIN {X 0,Y 474.629,Z 499.678,A -85,B 0,C 180,E1 -7440.885,E2 -7440.885} C_VEL
LIN {X 0,Y 474.682,Z 499.671,A -85,B 0,C 180,E1 -7442.62,E2 -7442.62} C_VEL
LIN {X 0,Y 474.085,Z 499.817,A -85,B 0,C 180,E1 -7443.328,E2 -7443.328} C_VEL
LIN {X 0,Y 471.313,Z 500.654,A -85,B 0,C 180,E1 -7444.477,E2 -7444.477} C_VEL
LIN {X 0,Y 468.938,Z 501.804,A -85,B 0,C 180,E1 -7445.397,E2 -7445.397} C_VEL
LIN {X 0,Y 467.92,Z 502.92,A -85,B 0,C 180,E1 -7446.102,E2 -7446.102} C_VEL
LIN {X 0,Y 467.841,Z 503.335,A -85,B 0,C 180,E1 -7446.339,E2 -7446.339} C_VEL
LIN {X 0,Y 467.787,Z 507.848,A -85,B 0,C 180,E1 -7448.864,E2 -7448.864} C_VEL
LIN {X 0,Y 467.738,Z 512.622,A -85,B 0,C 180,E1 -7451.606,E2 -7451.606} C_VEL
LIN {X 0,Y 467.693,Z 517.226,A -85,B 0,C 180,E1 -7454.306,E2 -7454.306} C_VEL
LIN {X 0,Y 467.599,Z 523.161,A -85,B 0,C 180,E1 -7457.852,E2 -7457.852} C_VEL
LIN {X 0,Y 467.525,Z 524.842,A -85,B 0,C 180,E1 -7458.783,E2 -7458.783} C_VEL
LIN {X 0,Y 470.716,Z 533.193,A -85,B 0,C 180,E1 -7459.12,E2 -7459.12} C_VEL
LIN {X 0,Y 475.321,Z 546.201,A -85,B 0,C 180,E1 -7459.702,E2 -7459.702} C_VEL
LIN {X 0,Y 477.123,Z 553.448,A -85,B 0,C 180,E1 -7460.026,E2 -7460.026} C_VEL
LIN {X 0,Y 476.44,Z 568.974,A -85,B 0,C 180,E1 -7460.578,E2 -7460.578} C_VEL
LIN {X 0,Y 475.591,Z 584.155,A -85,B 0,C 180,E1 -7461.287,E2 -7461.287} C_VEL
LIN {X 0,Y 474.639,Z 598.526,A -85,B 0,C 180,E1 -7462.127,E2 -7462.127} C_VEL
LIN {X 0,Y 473.557,Z 613.351,A -85,B 0,C 180,E1 -7463.181,E2 -7463.181} C_VEL
LIN {X 0,Y 472.442,Z 627.004,A -85,B 0,C 180,E1 -7464.343,E2 -7464.343} C_VEL
LIN {X 0,Y 471.432,Z 638.628,A -85,B 0,C 180,E1 -7465.51,E2 -7465.51} C_VEL
LIN {X 0,Y 470.462,Z 649.557,A -85,B 0,C 180,E1 -7466.788,E2 -7466.788} C_VEL
LIN {X 0,Y 469.522,Z 660.576,A -85,B 0,C 180,E1 -7468.284,E2 -7468.284} C_VEL
LIN {X 0,Y 468.578,Z 671.283,A -85,B 0,C 180,E1 -7469.999,E2 -7469.999} C_VEL
LIN {X 0,Y 467.986,Z 680.241,A -85,B 0,C 180,E1 -7471.72,E2 -7471.72} C_VEL
LIN {X 0,Y 467.401,Z 687.795,A -85,B 0,C 180,E1 -7473.447,E2 -7473.447} C_VEL
LIN {X 0,Y 467.12,Z 694.1,A -85,B 0,C 180,E1 -7475.178,E2 -7475.178} C_VEL
LIN {X 0,Y 466.893,Z 699.248,A -85,B 0,C 180,E1 -7476.915,E2 -7476.915} C_VEL
LIN {X 0,Y 466.725,Z 703.318,A -85,B 0,C 180,E1 -7478.66,E2 -7478.66} C_VEL
LIN {X 0,Y 466.623,Z 706.423,A -85,B 0,C 180,E1 -7480.412,E2 -7480.412} C_VEL
LIN {X 0,Y 466.603,Z 708.455,A -85,B 0,C 180,E1 -7482.172,E2 -7482.172} C_VEL
LIN {X 0,Y 466.499,Z 709.605,A -85,B 0,C 180,E1 -7483.947,E2 -7483.947} C_VEL
LIN {X 0,Y 466.501,Z 709.681,A -85,B 0,C 180,E1 -7485.733,E2 -7485.733} C_VEL
LIN {X 0,Y 466.517,Z 708.813,A -85,B 0,C 180,E1 -7487.534,E2 -7487.534} C_VEL
LIN {X 0,Y 466.542,Z 706.878,A -85,B 0,C 180,E1 -7489.353,E2 -7489.353} C_VEL
LIN {X 0,Y 466.696,Z 703.836,A -85,B 0,C 180,E1 -7491.186,E2 -7491.186} C_VEL
LIN {X 0,Y 466.841,Z 699.663,A -85,B 0,C 180,E1 -7493.041,E2 -7493.041} C_VEL
LIN {X 0,Y 467.133,Z 694.15,A -85,B 0,C 180,E1 -7494.913,E2 -7494.913} C_VEL
LIN {X 0,Y 467.517,Z 687.201,A -85,B 0,C 180,E1 -7496.805,E2 -7496.805} C_VEL
LIN {X 0,Y 468.085,Z 678.63,A -85,B 0,C 180,E1 -7498.714,E2 -7498.714} C_VEL
LIN {X 0,Y 468.801,Z 669.589,A -85,B 0,C 180,E1 -7500.394,E2 -7500.394} C_VEL
LIN {X 0,Y 469.565,Z 660.47,A -85,B 0,C 180,E1 -7501.841,E2 -7501.841} C_VEL
LIN {X 0,Y 470.524,Z 649.533,A -85,B 0,C 180,E1 -7503.322,E2 -7503.322} C_VEL
LIN {X 0,Y 471.57,Z 636.792,A -85,B 0,C 180,E1 -7504.793,E2 -7504.793} C_VEL
LIN {X 0,Y 472.764,Z 623.414,A -85,B 0,C 180,E1 -7506.088,E2 -7506.088} C_VEL
LIN {X 0,Y 473.832,Z 609.576,A -85,B 0,C 180,E1 -7507.219,E2 -7507.219} C_VEL
LIN {X 0,Y 474.924,Z 594.587,A -85,B 0,C 180,E1 -7508.229,E2 -7508.229} C_VEL
LIN {X 0,Y 475.886,Z 578.899,A -85,B 0,C 180,E1 -7509.079,E2 -7509.079} C_VEL
LIN {X 0,Y 476.686,Z 563.579,A -85,B 0,C 180,E1 -7509.73,E2 -7509.73} C_VEL
LIN {X 0,Y 477.052,Z 552.479,A -85,B 0,C 180,E1 -7510.109,E2 -7510.109} C_VEL
LIN {X 0,Y 473.439,Z 540.718,A -85,B 0,C 180,E1 -7510.655,E2 -7510.655} C_VEL
LIN {X 0,Y 467.549,Z 525.503,A -85,B 0,C 180,E1 -7511.31,E2 -7511.31} C_VEL
LIN {X 0,Y 467.48,Z 525.036,A -85,B 0,C 180,E1 -7511.338,E2 -7511.338} C_VEL
LIN {X 0,Y 467.556,Z 520.938,A -85,B 0,C 180,E1 -7513.821,E2 -7513.821} C_VEL
LIN {X 0,Y 467.666,Z 516.843,A -85,B 0,C 180,E1 -7516.268,E2 -7516.268} C_VEL
LIN {X 0,Y 467.801,Z 512.79,A -85,B 0,C 180,E1 -7518.69,E2 -7518.69} C_VEL
LIN {X 0,Y 467.84,Z 507.116,A -85,B 0,C 180,E1 -7521.981,E2 -7521.981} C_VEL
LIN {X 0,Y 467.903,Z 503.111,A -85,B 0,C 180,E1 -7524.2,E2 -7524.2} C_VEL
LIN {X 0,Y 467.628,Z 500.551,A -85,B 0,C 180,E1 -7525.748,E2 -7525.748} C_VEL
LIN {X 0,Y 467.567,Z 500.56,A -85,B 0,C 180,E1 -7529.265,E2 -7529.265} C_VEL
LIN {X 0,Y 467.637,Z 500.549,A -85,B 0,C 180,E1 -7532.458,E2 -7532.458} C_VEL
LIN {X 0,Y 467.605,Z 500.553,A -85,B 0,C 180,E1 -7535.112,E2 -7535.112} C_VEL
LIN {X 0,Y 467.534,Z 500.562,A -85,B 0,C 180,E1 -7537.926,E2 -7537.926} C_VEL
LIN {X 0,Y 467.615,Z 500.549,A -85,B 0,C 180,E1 -7540.691,E2 -7540.691} C_VEL
LIN {X 0,Y 467.639,Z 500.545,A -85,B 0,C 180,E1 -7544.114,E2 -7544.114} C_VEL
LIN {X 0,Y 467.673,Z 500.543,A -85,B 0,C 180,E1 -7547.855,E2 -7547.855} C_VEL
LIN {X 0,Y 467.673,Z 500.541,A -85,B 0,C 180,E1 -7551.357,E2 -7551.357} C_VEL
LIN {X 0,Y 467.744,Z 500.535,A -85,B 0,C 180,E1 -7553.962,E2 -7553.962} C_VEL
LIN {X 0,Y 467.852,Z 500.52,A -85,B 0,C 180,E1 -7557.417,E2 -7557.417} C_VEL
LIN {X 0,Y 467.872,Z 500.518,A -85,B 0,C 180,E1 -7560,E2 -7560} C_VEL
LIN {X 0,Y 467.851,Z 500.518,A -85,B 0,C 180,E1 -7562.583,E2 -7562.583} C_VEL
LIN {X 0,Y 467.733,Z 500.531,A -85,B 0,C 180,E1 -7566.037,E2 -7566.037} C_VEL
LIN {X 0,Y 467.671,Z 500.539,A -85,B 0,C 180,E1 -7568.643,E2 -7568.643} C_VEL
LIN {X 0,Y 467.679,Z 500.536,A -85,B 0,C 180,E1 -7572.379,E2 -7572.379} C_VEL
LIN {X 0,Y 467.637,Z 500.539,A -85,B 0,C 180,E1 -7575.885,E2 -7575.885} C_VEL
LIN {X 0,Y 467.613,Z 500.541,A -85,B 0,C 180,E1 -7579.308,E2 -7579.308} C_VEL
LIN {X 0,Y 467.556,Z 500.558,A -85,B 0,C 180,E1 -7582.072,E2 -7582.072} C_VEL
LIN {X 0,Y 467.602,Z 500.53,A -85,B 0,C 180,E1 -7584.887,E2 -7584.887} C_VEL
LIN {X 0,Y 467.617,Z 500.552,A -85,B 0,C 180,E1 -7587.769,E2 -7587.769} C_VEL
LIN {X 0,Y 467.562,Z 500.557,A -85,B 0,C 180,E1 -7591.046,E2 -7591.046} C_VEL
LIN {X 0,Y 467.579,Z 500.554,A -85,B 0,C 180,E1 -7594.243,E2 -7594.243} C_VEL
LIN {X 0,Y 467.543,Z 500.559,A -85,B 0,C 180,E1 -7597.188,E2 -7597.188} C_VEL
LIN {X 0,Y 467.592,Z 500.553,A -85,B 0,C 180,E1 -7600.263,E2 -7600.263} C_VEL
LIN {X 0,Y 467.626,Z 500.628,A -85,B 0,C 180,E1 -7602.621,E2 -7602.621} C_VEL
LIN {X 0,Y 469.763,Z 510.515,A -85,B 0,C 180,E1 -7605.899,E2 -7605.899} C_VEL
LIN {X 0,Y 471.63,Z 519.103,A -85,B 0,C 180,E1 -7608.625,E2 -7608.625} C_VEL
LIN {X 0,Y 472.042,Z 524.428,A -85,B 0,C 180,E1 -7610.195,E2 -7610.195} C_VEL
LIN {X 0,Y 471.324,Z 536.872,A -85,B 0,C 180,E1 -7613.629,E2 -7613.629} C_VEL
LIN {X 0,Y 470.622,Z 549.972,A -85,B 0,C 180,E1 -7617.107,E2 -7617.107} C_VEL
LIN {X 0,Y 470.003,Z 563.028,A -85,B 0,C 180,E1 -7620.434,E2 -7620.434} C_VEL
LIN {X 0,Y 469.488,Z 574.571,A -85,B 0,C 180,E1 -7623.316,E2 -7623.316} C_VEL
LIN {X 0,Y 469.429,Z 576.561,A -85,B 0,C 180,E1 -7623.757,E2 -7623.757} C_VEL
LIN {X 0,Y 475.547,Z 598.331,A -85,B 0,C 180,E1 -7624.529,E2 -7624.529} C_VEL
LIN {X 0,Y 477.168,Z 605.145,A -85,B 0,C 180,E1 -7624.796,E2 -7624.796} C_VEL
LIN {X 0,Y 476.497,Z 621.835,A -85,B 0,C 180,E1 -7625.336,E2 -7625.336} C_VEL
LIN {X 0,Y 475.612,Z 637.783,A -85,B 0,C 180,E1 -7626.025,E2 -7626.025} C_VEL
LIN {X 0,Y 474.682,Z 652.455,A -85,B 0,C 180,E1 -7626.83,E2 -7626.83} C_VEL
LIN {X 0,Y 473.61,Z 666.578,A -85,B 0,C 180,E1 -7627.767,E2 -7627.767} C_VEL
LIN {X 0,Y 472.487,Z 681.49,A -85,B 0,C 180,E1 -7628.972,E2 -7628.972} C_VEL
LIN {X 0,Y 471.291,Z 695.102,A -85,B 0,C 180,E1 -7630.288,E2 -7630.288} C_VEL
LIN {X 0,Y 470.243,Z 707.511,A -85,B 0,C 180,E1 -7631.709,E2 -7631.709} C_VEL
LIN {X 0,Y 469.309,Z 718.943,A -85,B 0,C 180,E1 -7633.247,E2 -7633.247} C_VEL
LIN {X 0,Y 468.587,Z 728.745,A -85,B 0,C 180,E1 -7634.784,E2 -7634.784} C_VEL
LIN {X 0,Y 467.873,Z 738.17,A -85,B 0,C 180,E1 -7636.537,E2 -7636.537} C_VEL
LIN {X 0,Y 467.431,Z 746.052,A -85,B 0,C 180,E1 -7638.29,E2 -7638.29} C_VEL
LIN {X 0,Y 467.024,Z 752.628,A -85,B 0,C 180,E1 -7640.035,E2 -7640.035} C_VEL
LIN {X 0,Y 466.858,Z 757.959,A -85,B 0,C 180,E1 -7641.779,E2 -7641.779} C_VEL
LIN {X 0,Y 466.756,Z 762.335,A -85,B 0,C 180,E1 -7643.598,E2 -7643.598} C_VEL
LIN {X 0,Y 466.607,Z 765.979,A -85,B 0,C 180,E1 -7645.682,E2 -7645.682} C_VEL
LIN {X 0,Y 466.635,Z 767.897,A -85,B 0,C 180,E1 -7647.411,E2 -7647.411} C_VEL
LIN {X 0,Y 466.586,Z 768.848,A -85,B 0,C 180,E1 -7649.138,E2 -7649.138} C_VEL
LIN {X 0,Y 466.586,Z 768.847,A -85,B 0,C 180,E1 -7650.864,E2 -7650.864} C_VEL
LIN {X 0,Y 466.635,Z 767.895,A -85,B 0,C 180,E1 -7652.591,E2 -7652.591} C_VEL
LIN {X 0,Y 466.607,Z 765.975,A -85,B 0,C 180,E1 -7654.32,E2 -7654.32} C_VEL
LIN {X 0,Y 466.758,Z 762.333,A -85,B 0,C 180,E1 -7656.404,E2 -7656.404} C_VEL
LIN {X 0,Y 466.86,Z 757.958,A -85,B 0,C 180,E1 -7658.223,E2 -7658.223} C_VEL
LIN {X 0,Y 467.024,Z 752.623,A -85,B 0,C 180,E1 -7659.966,E2 -7659.966} C_VEL
LIN {X 0,Y 467.428,Z 746.045,A -85,B 0,C 180,E1 -7661.712,E2 -7661.712} C_VEL
LIN {X 0,Y 467.876,Z 738.161,A -85,B 0,C 180,E1 -7663.464,E2 -7663.464} C_VEL
LIN {X 0,Y 468.586,Z 728.735,A -85,B 0,C 180,E1 -7665.217,E2 -7665.217} C_VEL
LIN {X 0,Y 469.475,Z 717.445,A -85,B 0,C 180,E1 -7666.973,E2 -7666.973} C_VEL
LIN {X 0,Y 470.403,Z 705.714,A -85,B 0,C 180,E1 -7668.511,E2 -7668.511} C_VEL
LIN {X 0,Y 471.378,Z 693.967,A -85,B 0,C 180,E1 -7669.828,E2 -7669.828} C_VEL
LIN {X 0,Y 472.461,Z 681.469,A -85,B 0,C 180,E1 -7671.031,E2 -7671.031} C_VEL
LIN {X 0,Y 473.597,Z 666.55,A -85,B 0,C 180,E1 -7672.236,E2 -7672.236} C_VEL
LIN {X 0,Y 474.733,Z 651.343,A -85,B 0,C 180,E1 -7673.239,E2 -7673.239} C_VEL
LIN {X 0,Y 475.679,Z 636.604,A -85,B 0,C 180,E1 -7674.031,E2 -7674.031} C_VEL
LIN {X 0,Y 476.504,Z 620.233,A -85,B 0,C 180,E1 -7674.719,E2 -7674.719} C_VEL
LIN {X 0,Y 477.081,Z 604.563,A -85,B 0,C 180,E1 -7675.218,E2 -7675.218} C_VEL
LIN {X 0,Y 471.785,Z 585.065,A -85,B 0,C 180,E1 -7675.947,E2 -7675.947} C_VEL
LIN {X 0,Y 469.52,Z 576.698,A -85,B 0,C 180,E1 -7676.225,E2 -7676.225} C_VEL
LIN {X 0,Y 469.299,Z 575.014,A -85,B 0,C 180,E1 -7676.275,E2 -7676.275} C_VEL
LIN {X 0,Y 469.698,Z 561.524,A -85,B 0,C 180,E1 -7679.343,E2 -7679.343} C_VEL
LIN {X 0,Y 469.991,Z 548.59,A -85,B 0,C 180,E1 -7682.317,E2 -7682.317} C_VEL
LIN {X 0,Y 470.321,Z 535.552,A -85,B 0,C 180,E1 -7685.387,E2 -7685.387} C_VEL
LIN {X 0,Y 470.574,Z 522.657,A -85,B 0,C 180,E1 -7688.575,E2 -7688.575} C_VEL
LIN {X 0,Y 470.597,Z 515.794,A -85,B 0,C 180,E1 -7690.391,E2 -7690.391} C_VEL
LIN {X 0,Y 469.147,Z 507.977,A -85,B 0,C 180,E1 -7692.774,E2 -7692.774} C_VEL
LIN {X 0,Y 467.832,Z 501.626,A -85,B 0,C 180,E1 -7695.086,E2 -7695.086} C_VEL
LIN {X 0,Y 467.584,Z 500.555,A -85,B 0,C 180,E1 -7695.581,E2 -7695.581} C_VEL
LIN {X 0,Y 467.583,Z 500.556,A -85,B 0,C 180,E1 -7698.723,E2 -7698.723} C_VEL
LIN {X 0,Y 467.567,Z 500.557,A -85,B 0,C 180,E1 -7701.956,E2 -7701.956} C_VEL
LIN {X 0,Y 467.569,Z 500.556,A -85,B 0,C 180,E1 -7705.168,E2 -7705.168} C_VEL
LIN {X 0,Y 467.584,Z 500.556,A -85,B 0,C 180,E1 -7708.26,E2 -7708.26} C_VEL
LIN {X 0,Y 467.578,Z 500.555,A -85,B 0,C 180,E1 -7711.251,E2 -7711.251} C_VEL
LIN {X 0,Y 467.618,Z 500.55,A -85,B 0,C 180,E1 -7713.2,E2 -7713.2} C_VEL
LIN {X 0,Y 467.633,Z 500.55,A -85,B 0,C 180,E1 -7714.299,E2 -7714.299} C_VEL
LIN {X 0,Y 468.622,Z 503.393,A -85,B 0,C 180,E1 -7714.431,E2 -7714.431} C_VEL
LIN {X 0,Y 474.496,Z 517.38,A -85,B 0,C 180,E1 -7715.186,E2 -7715.186} C_VEL
LIN {X 0,Y 476.216,Z 522.447,A -85,B 0,C 180,E1 -7715.459,E2 -7715.459} C_VEL
LIN {X 0,Y 475.585,Z 539.212,A -85,B 0,C 180,E1 -7716.148,E2 -7716.148} C_VEL
LIN {X 0,Y 474.694,Z 554.174,A -85,B 0,C 180,E1 -7716.927,E2 -7716.927} C_VEL
LIN {X 0,Y 473.85,Z 567.613,A -85,B 0,C 180,E1 -7717.778,E2 -7717.778} C_VEL
LIN {X 0,Y 472.913,Z 582.012,A -85,B 0,C 180,E1 -7718.877,E2 -7718.877} C_VEL
LIN {X 0,Y 471.885,Z 595.257,A -85,B 0,C 180,E1 -7720.082,E2 -7720.082} C_VEL
LIN {X 0,Y 470.837,Z 608.339,A -85,B 0,C 180,E1 -7721.507,E2 -7721.507} C_VEL
LIN {X 0,Y 469.922,Z 619.274,A -85,B 0,C 180,E1 -7722.918,E2 -7722.918} C_VEL
LIN {X 0,Y 469.092,Z 630.153,A -85,B 0,C 180,E1 -7724.578,E2 -7724.578} C_VEL
LIN {X 0,Y 468.331,Z 639.767,A -85,B 0,C 180,E1 -7726.329,E2 -7726.329} C_VEL
LIN {X 0,Y 467.919,Z 646.859,A -85,B 0,C 180,E1 -7727.862,E2 -7727.862} C_VEL
LIN {X 0,Y 467.368,Z 653.569,A -85,B 0,C 180,E1 -7729.604,E2 -7729.604} C_VEL
LIN {X 0,Y 467.119,Z 659.06,A -85,B 0,C 180,E1 -7731.347,E2 -7731.347} C_VEL
LIN {X 0,Y 466.968,Z 664.039,A -85,B 0,C 180,E1 -7733.374,E2 -7733.374} C_VEL
LIN {X 0,Y 466.736,Z 667.987,A -85,B 0,C 180,E1 -7735.683,E2 -7735.683} C_VEL
LIN {X 0,Y 466.703,Z 669.814,A -85,B 0,C 180,E1 -7737.411,E2 -7737.411} C_VEL
LIN {X 0,Y 466.653,Z 670.728,A -85,B 0,C 180,E1 -7739.137,E2 -7739.137} C_VEL
LIN {X 0,Y 466.649,Z 670.701,A -85,B 0,C 180,E1 -7740.863,E2 -7740.863} C_VEL
LIN {X 0,Y 466.7,Z 669.777,A -85,B 0,C 180,E1 -7742.59,E2 -7742.59} C_VEL
LIN {X 0,Y 466.718,Z 667.879,A -85,B 0,C 180,E1 -7744.318,E2 -7744.318} C_VEL
LIN {X 0,Y 466.834,Z 665.044,A -85,B 0,C 180,E1 -7746.05,E2 -7746.05} C_VEL
LIN {X 0,Y 466.991,Z 661.179,A -85,B 0,C 180,E1 -7747.785,E2 -7747.785} C_VEL
LIN {X 0,Y 467.159,Z 656.203,A -85,B 0,C 180,E1 -7749.526,E2 -7749.526} C_VEL
LIN {X 0,Y 467.49,Z 650.083,A -85,B 0,C 180,E1 -7751.271,E2 -7751.271} C_VEL
LIN {X 0,Y 467.957,Z 642.592,A -85,B 0,C 180,E1 -7753.02,E2 -7753.02} C_VEL
LIN {X 0,Y 468.627,Z 633.565,A -85,B 0,C 180,E1 -7754.771,E2 -7754.771} C_VEL
LIN {X 0,Y 469.443,Z 622.783,A -85,B 0,C 180,E1 -7756.526,E2 -7756.526} C_VEL
LIN {X 0,Y 470.313,Z 611.577,A -85,B 0,C 180,E1 -7758.064,E2 -7758.064} C_VEL
LIN {X 0,Y 471.301,Z 599.324,A -85,B 0,C 180,E1 -7759.491,E2 -7759.491} C_VEL
LIN {X 0,Y 472.403,Z 586.041,A -85,B 0,C 180,E1 -7760.795,E2 -7760.795} C_VEL
LIN {X 0,Y 473.407,Z 572.627,A -85,B 0,C 180,E1 -7761.901,E2 -7761.901} C_VEL
LIN {X 0,Y 474.468,Z 558.236,A -85,B 0,C 180,E1 -7762.895,E2 -7762.895} C_VEL
LIN {X 0,Y 475.306,Z 544.283,A -85,B 0,C 180,E1 -7763.702,E2 -7763.702} C_VEL
LIN {X 0,Y 476.159,Z 527.438,A -85,B 0,C 180,E1 -7764.475,E2 -7764.475} C_VEL
LIN {X 0,Y 476.361,Z 522.029,A -85,B 0,C 180,E1 -7764.677,E2 -7764.677} C_VEL
LIN {X 0,Y 469.962,Z 506.349,A -85,B 0,C 180,E1 -7765.557,E2 -7765.557} C_VEL
LIN {X 0,Y 467.671,Z 500.933,A -85,B 0,C 180,E1 -7765.837,E2 -7765.837} C_VEL
LIN {X 0,Y 467.612,Z 500.55,A -85,B 0,C 180,E1 -7765.87,E2 -7765.87} C_VEL
LIN {X 0,Y 467.581,Z 500.555,A -85,B 0,C 180,E1 -7768.75,E2 -7768.75} C_VEL
LIN {X 0,Y 467.587,Z 500.556,A -85,B 0,C 180,E1 -7771.74,E2 -7771.74} C_VEL
LIN {X 0,Y 467.573,Z 500.557,A -85,B 0,C 180,E1 -7774.832,E2 -7774.832} C_VEL
LIN {X 0,Y 467.571,Z 500.555,A -85,B 0,C 180,E1 -7778.045,E2 -7778.045} C_VEL
LIN {X 0,Y 467.583,Z 500.554,A -85,B 0,C 180,E1 -7781.277,E2 -7781.277} C_VEL
LIN {X 0,Y 467.557,Z 500.556,A -85,B 0,C 180,E1 -7783.821,E2 -7783.821} C_VEL
LIN {X 0,Y 467.559,Z 500.558,A -85,B 0,C 180,E1 -7786.255,E2 -7786.255} C_VEL
LIN {X 0,Y 467.584,Z 500.555,A -85,B 0,C 180,E1 -7788.723,E2 -7788.723} C_VEL
LIN {X 0,Y 467.57,Z 500.558,A -85,B 0,C 180,E1 -7791.955,E2 -7791.955} C_VEL
LIN {X 0,Y 467.57,Z 500.556,A -85,B 0,C 180,E1 -7795.167,E2 -7795.167} C_VEL
LIN {X 0,Y 467.589,Z 500.557,A -85,B 0,C 180,E1 -7798.26,E2 -7798.26} C_VEL
LIN {X 0,Y 467.582,Z 500.556,A -85,B 0,C 180,E1 -7801.25,E2 -7801.25} C_VEL
LIN {X 0,Y 467.679,Z 500.545,A -85,B 0,C 180,E1 -7804.376,E2 -7804.376} C_VEL
LIN {X 0,Y 467.774,Z 500.766,A -85,B 0,C 180,E1 -7804.905,E2 -7804.905} C_VEL
LIN {X 0,Y 467.841,Z 503.335,A -85,B 0,C 180,E1 -7806.339,E2 -7806.339} C_VEL
LIN {X 0,Y 467.176,Z 504.705,A -85,B 0,C 180,E1 -7807.038,E2 -7807.038} C_VEL
LIN {X 0,Y 464.298,Z 507.177,A -85,B 0,C 180,E1 -7808.165,E2 -7808.165} C_VEL
LIN {X 0,Y 461.86,Z 509.171,A -85,B 0,C 180,E1 -7809.073,E2 -7809.073} C_VEL
LIN {X 0,Y 460.815,Z 510.562,A -85,B 0,C 180,E1 -7809.779,E2 -7809.779} C_VEL
LIN {X 0,Y 460.732,Z 510.99,A -85,B 0,C 180,E1 -7810.019,E2 -7810.019} C_VEL
LIN {X 0,Y 460.683,Z 516.363,A -85,B 0,C 180,E1 -7813.15,E2 -7813.15} C_VEL
LIN {X 0,Y 460.59,Z 520.951,A -85,B 0,C 180,E1 -7815.868,E2 -7815.868} C_VEL
LIN {X 0,Y 460.543,Z 525.055,A -85,B 0,C 180,E1 -7818.337,E2 -7818.337} C_VEL
LIN {X 0,Y 462.276,Z 530.101,A -85,B 0,C 180,E1 -7818.552,E2 -7818.552} C_VEL
LIN {X 0,Y 468.464,Z 546.398,A -85,B 0,C 180,E1 -7819.302,E2 -7819.302} C_VEL
LIN {X 0,Y 470.665,Z 555.075,A -85,B 0,C 180,E1 -7819.703,E2 -7819.703} C_VEL
LIN {X 0,Y 469.851,Z 571.646,A -85,B 0,C 180,E1 -7820.321,E2 -7820.321} C_VEL
LIN {X 0,Y 468.974,Z 586.701,A -85,B 0,C 180,E1 -7821.055,E2 -7821.055} C_VEL
LIN {X 0,Y 467.979,Z 600.719,A -85,B 0,C 180,E1 -7821.906,E2 -7821.906} C_VEL
LIN {X 0,Y 466.833,Z 615.224,A -85,B 0,C 180,E1 -7822.973,E2 -7822.973} C_VEL
LIN {X 0,Y 465.657,Z 628.636,A -85,B 0,C 180,E1 -7824.152,E2 -7824.152} C_VEL
LIN {X 0,Y 464.533,Z 641.096,A -85,B 0,C 180,E1 -7825.443,E2 -7825.443} C_VEL
LIN {X 0,Y 463.392,Z 653.435,A -85,B 0,C 180,E1 -7826.956,E2 -7826.956} C_VEL
LIN {X 0,Y 462.452,Z 663.89,A -85,B 0,C 180,E1 -7828.475,E2 -7828.475} C_VEL
LIN {X 0,Y 461.488,Z 674.118,A -85,B 0,C 180,E1 -7830.217,E2 -7830.217} C_VEL
LIN {X 0,Y 460.949,Z 681.766,A -85,B 0,C 180,E1 -7831.746,E2 -7831.746} C_VEL
LIN {X 0,Y 460.362,Z 689.143,A -85,B 0,C 180,E1 -7833.5,E2 -7833.5} C_VEL
LIN {X 0,Y 460.076,Z 695.258,A -85,B 0,C 180,E1 -7835.258,E2 -7835.258} C_VEL
LIN {X 0,Y 459.825,Z 700.313,A -85,B 0,C 180,E1 -7837.022,E2 -7837.022} C_VEL
LIN {X 0,Y 459.646,Z 704.22,A -85,B 0,C 180,E1 -7838.794,E2 -7838.794} C_VEL
LIN {X 0,Y 459.554,Z 707.182,A -85,B 0,C 180,E1 -7840.574,E2 -7840.574} C_VEL
LIN {X 0,Y 459.508,Z 709.111,A -85,B 0,C 180,E1 -7842.363,E2 -7842.363} C_VEL
LIN {X 0,Y 459.418,Z 710.096,A -85,B 0,C 180,E1 -7844.167,E2 -7844.167} C_VEL
LIN {X 0,Y 459.404,Z 710.092,A -85,B 0,C 180,E1 -7845.983,E2 -7845.983} C_VEL
LIN {X 0,Y 459.457,Z 709.053,A -85,B 0,C 180,E1 -7847.813,E2 -7847.813} C_VEL
LIN {X 0,Y 459.48,Z 707.031,A -85,B 0,C 180,E1 -7849.663,E2 -7849.663} C_VEL
LIN {X 0,Y 459.661,Z 703.81,A -85,B 0,C 180,E1 -7851.526,E2 -7851.526} C_VEL
LIN {X 0,Y 459.844,Z 699.19,A -85,B 0,C 180,E1 -7853.506,E2 -7853.506} C_VEL
LIN {X 0,Y 460.17,Z 693.805,A -85,B 0,C 180,E1 -7855.316,E2 -7855.316} C_VEL
LIN {X 0,Y 460.609,Z 686.656,A -85,B 0,C 180,E1 -7857.24,E2 -7857.24} C_VEL
LIN {X 0,Y 461.163,Z 679.022,A -85,B 0,C 180,E1 -7858.936,E2 -7858.936} C_VEL
LIN {X 0,Y 461.912,Z 669.96,A -85,B 0,C 180,E1 -7860.643,E2 -7860.643} C_VEL
LIN {X 0,Y 462.904,Z 659.164,A -85,B 0,C 180,E1 -7862.355,E2 -7862.355} C_VEL
LIN {X 0,Y 464.003,Z 647.556,A -85,B 0,C 180,E1 -7863.908,E2 -7863.908} C_VEL
LIN {X 0,Y 465.088,Z 635.132,A -85,B 0,C 180,E1 -7865.313,E2 -7865.313} C_VEL
LIN {X 0,Y 466.263,Z 622.309,A -85,B 0,C 180,E1 -7866.538,E2 -7866.538} C_VEL
LIN {X 0,Y 467.472,Z 607.19,A -85,B 0,C 180,E1 -7867.751,E2 -7867.751} C_VEL
LIN {X 0,Y 468.621,Z 591.932,A -85,B 0,C 180,E1 -7868.752,E2 -7868.752} C_VEL
LIN {X 0,Y 469.605,Z 576.578,A -85,B 0,C 180,E1 -7869.565,E2 -7869.565} C_VEL
LIN {X 0,Y 470.419,Z 560.795,A -85,B 0,C 180,E1 -7870.214,E2 -7870.214} C_VEL
LIN {X 0,Y 470.628,Z 554.134,A -85,B 0,C 180,E1 -7870.435,E2 -7870.435} C_VEL
LIN {X 0,Y 467.203,Z 542.994,A -85,B 0,C 180,E1 -7870.978,E2 -7870.978} C_VEL
LIN {X 0,Y 460.634,Z 526.27,A -85,B 0,C 180,E1 -7871.742,E2 -7871.742} C_VEL
LIN {X 0,Y 460.464,Z 525.477,A -85,B 0,C 180,E1 -7871.787,E2 -7871.787} C_VEL
LIN {X 0,Y 460.576,Z 520.871,A -85,B 0,C 180,E1 -7874.579,E2 -7874.579} C_VEL
LIN {X 0,Y 460.746,Z 515.426,A -85,B 0,C 180,E1 -7877.843,E2 -7877.843} C_VEL
LIN {X 0,Y 460.835,Z 510.023,A -85,B 0,C 180,E1 -7881.055,E2 -7881.055} C_VEL
LIN {X 0,Y 460.93,Z 504.955,A -85,B 0,C 180,E1 -7883.909,E2 -7883.909} C_VEL
LIN {X 0,Y 460.581,Z 501.43,A -85,B 0,C 180,E1 -7885.957,E2 -7885.957} C_VEL
LIN {X 0,Y 460.529,Z 501.437,A -85,B 0,C 180,E1 -7888.743,E2 -7888.743} C_VEL
LIN {X 0,Y 460.55,Z 501.431,A -85,B 0,C 180,E1 -7891.766,E2 -7891.766} C_VEL
LIN {X 0,Y 460.574,Z 501.428,A -85,B 0,C 180,E1 -7894.706,E2 -7894.706} C_VEL
LIN {X 0,Y 460.507,Z 501.438,A -85,B 0,C 180,E1 -7897.571,E2 -7897.571} C_VEL
LIN {X 0,Y 460.56,Z 501.43,A -85,B 0,C 180,E1 -7900.384,E2 -7900.384} C_VEL
LIN {X 0,Y 460.556,Z 501.428,A -85,B 0,C 180,E1 -7903.145,E2 -7903.145} C_VEL
LIN {X 0,Y 460.545,Z 501.429,A -85,B 0,C 180,E1 -7905.867,E2 -7905.867} C_VEL
LIN {X 0,Y 460.622,Z 501.419,A -85,B 0,C 180,E1 -7908.559,E2 -7908.559} C_VEL
LIN {X 0,Y 460.684,Z 501.409,A -85,B 0,C 180,E1 -7912.108,E2 -7912.108} C_VEL
LIN {X 0,Y 460.697,Z 501.41,A -85,B 0,C 180,E1 -7914.748,E2 -7914.748} C_VEL
LIN {X 0,Y 460.817,Z 501.396,A -85,B 0,C 180,E1 -7917.377,E2 -7917.377} C_VEL
LIN {X 0,Y 460.843,Z 501.394,A -85,B 0,C 180,E1 -7920,E2 -7920} C_VEL
LIN {X 0,Y 460.816,Z 501.395,A -85,B 0,C 180,E1 -7922.622,E2 -7922.622} C_VEL
LIN {X 0,Y 460.699,Z 501.408,A -85,B 0,C 180,E1 -7926.13,E2 -7926.13} C_VEL
LIN {X 0,Y 460.619,Z 501.416,A -85,B 0,C 180,E1 -7928.776,E2 -7928.776} C_VEL
LIN {X 0,Y 460.622,Z 501.415,A -85,B 0,C 180,E1 -7932.457,E2 -7932.457} C_VEL
LIN {X 0,Y 460.588,Z 501.416,A -85,B 0,C 180,E1 -7935.998,E2 -7935.998} C_VEL
LIN {X 0,Y 460.559,Z 501.415,A -85,B 0,C 180,E1 -7938.902,E2 -7938.902} C_VEL
LIN {X 0,Y 460.552,Z 501.43,A -85,B 0,C 180,E1 -7941.483,E2 -7941.483} C_VEL
LIN {X 0,Y 460.536,Z 501.408,A -85,B 0,C 180,E1 -7944.332,E2 -7944.332} C_VEL
LIN {X 0,Y 460.573,Z 501.426,A -85,B 0,C 180,E1 -7947.243,E2 -7947.243} C_VEL
LIN {X 0,Y 460.516,Z 501.435,A -85,B 0,C 180,E1 -7950.239,E2 -7950.239} C_VEL
LIN {X 0,Y 460.519,Z 501.435,A -85,B 0,C 180,E1 -7953.325,E2 -7953.325} C_VEL
LIN {X 0,Y 460.47,Z 501.438,A -85,B 0,C 180,E1 -7956.53,E2 -7956.53} C_VEL
LIN {X 0,Y 460.575,Z 501.426,A -85,B 0,C 180,E1 -7959.857,E2 -7959.857} C_VEL
LIN {X 0,Y 460.578,Z 501.542,A -85,B 0,C 180,E1 -7962.175,E2 -7962.175} C_VEL
LIN {X 0,Y 462.391,Z 509.796,A -85,B 0,C 180,E1 -7964.972,E2 -7964.972} C_VEL
LIN {X 0,Y 464.319,Z 518.728,A -85,B 0,C 180,E1 -7967.874,E2 -7967.874} C_VEL
LIN {X 0,Y 465.128,Z 523.93,A -85,B 0,C 180,E1 -7969.481,E2 -7969.481} C_VEL
LIN {X 0,Y 464.931,Z 529.75,A -85,B 0,C 180,E1 -7971.149,E2 -7971.149} C_VEL
LIN {X 0,Y 464.26,Z 541.286,A -85,B 0,C 180,E1 -7974.353,E2 -7974.353} C_VEL
LIN {X 0,Y 463.621,Z 552.857,A -85,B 0,C 180,E1 -7977.444,E2 -7977.444} C_VEL
LIN {X 0,Y 462.936,Z 566.409,A -85,B 0,C 180,E1 -7980.936,E2 -7980.936} C_VEL
LIN {X 0,Y 462.46,Z 575.811,A -85,B 0,C 180,E1 -7983.317,E2 -7983.317} C_VEL
LIN {X 0,Y 468.344,Z 597.042,A -85,B 0,C 180,E1 -7984.09,E2 -7984.09} C_VEL
LIN {X 0,Y 470.627,Z 606.878,A -85,B 0,C 180,E1 -7984.495,E2 -7984.495} C_VEL
LIN {X 0,Y 469.92,Z 622.846,A -85,B 0,C 180,E1 -7985.036,E2 -7985.036} C_VEL
LIN {X 0,Y 468.927,Z 639.362,A -85,B 0,C 180,E1 -7985.779,E2 -7985.779} C_VEL
LIN {X 0,Y 467.956,Z 653.563,A -85,B 0,C 180,E1 -7986.585,E2 -7986.585} C_VEL
LIN {X 0,Y 466.703,Z 669.152,A -85,B 0,C 180,E1 -7987.653,E2 -7987.653} C_VEL
LIN {X 0,Y 465.679,Z 682.672,A -85,B 0,C 180,E1 -7988.766,E2 -7988.766} C_VEL
LIN {X 0,Y 464.435,Z 696.53,A -85,B 0,C 180,E1 -7990.14,E2 -7990.14} C_VEL
LIN {X 0,Y 463.27,Z 709.292,A -85,B 0,C 180,E1 -7991.653,E2 -7991.653} C_VEL
LIN {X 0,Y 462.246,Z 721.044,A -85,B 0,C 180,E1 -7993.305,E2 -7993.305} C_VEL
LIN {X 0,Y 461.401,Z 731.211,A -85,B 0,C 180,E1 -7994.994,E2 -7994.994} C_VEL
LIN {X 0,Y 460.732,Z 740.272,A -85,B 0,C 180,E1 -7996.774,E2 -7996.774} C_VEL
LIN {X 0,Y 460.299,Z 747.859,A -85,B 0,C 180,E1 -7998.553,E2 -7998.553} C_VEL
LIN {X 0,Y 459.857,Z 755.468,A -85,B 0,C 180,E1 -8000.767,E2 -8000.767} C_VEL
LIN {X 0,Y 459.722,Z 761.252,A -85,B 0,C 180,E1 -8002.976,E2 -8002.976} C_VEL
LIN {X 0,Y 459.582,Z 764.635,A -85,B 0,C 180,E1 -8004.737,E2 -8004.737} C_VEL
LIN {X 0,Y 459.533,Z 767.092,A -85,B 0,C 180,E1 -8006.494,E2 -8006.494} C_VEL
LIN {X 0,Y 459.511,Z 768.478,A -85,B 0,C 180,E1 -8008.248,E2 -8008.248} C_VEL
LIN {X 0,Y 459.469,Z 769,A -85,B 0,C 180,E1 -8010.001,E2 -8010.001} C_VEL
LIN {X 0,Y 459.512,Z 768.477,A -85,B 0,C 180,E1 -8011.754,E2 -8011.754} C_VEL
LIN {X 0,Y 459.534,Z 767.088,A -85,B 0,C 180,E1 -8013.508,E2 -8013.508} C_VEL
LIN {X 0,Y 459.583,Z 764.632,A -85,B 0,C 180,E1 -8015.265,E2 -8015.265} C_VEL
LIN {X 0,Y 459.723,Z 761.25,A -85,B 0,C 180,E1 -8017.026,E2 -8017.026} C_VEL
LIN {X 0,Y 459.858,Z 755.465,A -85,B 0,C 180,E1 -8019.235,E2 -8019.235} C_VEL
LIN {X 0,Y 460.268,Z 747.852,A -85,B 0,C 180,E1 -8021.45,E2 -8021.45} C_VEL
LIN {X 0,Y 460.735,Z 740.263,A -85,B 0,C 180,E1 -8023.228,E2 -8023.228} C_VEL
LIN {X 0,Y 461.398,Z 731.202,A -85,B 0,C 180,E1 -8025.008,E2 -8025.008} C_VEL
LIN {X 0,Y 462.253,Z 721.025,A -85,B 0,C 180,E1 -8026.698,E2 -8026.698} C_VEL
LIN {X 0,Y 463.278,Z 709.276,A -85,B 0,C 180,E1 -8028.348,E2 -8028.348} C_VEL
LIN {X 0,Y 464.39,Z 696.389,A -85,B 0,C 180,E1 -8029.878,E2 -8029.878} C_VEL
LIN {X 0,Y 465.651,Z 682.649,A -85,B 0,C 180,E1 -8031.238,E2 -8031.238} C_VEL
LIN {X 0,Y 466.724,Z 668.998,A -85,B 0,C 180,E1 -8032.348,E2 -8032.348} C_VEL
LIN {X 0,Y 467.931,Z 653.102,A -85,B 0,C 180,E1 -8033.419,E2 -8033.419} C_VEL
LIN {X 0,Y 468.935,Z 637.459,A -85,B 0,C 180,E1 -8034.282,E2 -8034.282} C_VEL
LIN {X 0,Y 469.847,Z 621.949,A -85,B 0,C 180,E1 -8034.967,E2 -8034.967} C_VEL
LIN {X 0,Y 470.422,Z 605.79,A -85,B 0,C 180,E1 -8035.513,E2 -8035.513} C_VEL
LIN {X 0,Y 465.991,Z 588.973,A -85,B 0,C 180,E1 -8036.186,E2 -8036.186} C_VEL
LIN {X 0,Y 463.348,Z 579.013,A -85,B 0,C 180,E1 -8036.55,E2 -8036.55} C_VEL
LIN {X 0,Y 462.299,Z 573.725,A -85,B 0,C 180,E1 -8036.705,E2 -8036.705} C_VEL
LIN {X 0,Y 462.704,Z 560.364,A -85,B 0,C 180,E1 -8039.795,E2 -8039.795} C_VEL
LIN {X 0,Y 463.003,Z 547.291,A -85,B 0,C 180,E1 -8042.865,E2 -8042.865} C_VEL
LIN {X 0,Y 463.386,Z 534.368,A -85,B 0,C 180,E1 -8045.995,E2 -8045.995} C_VEL
LIN {X 0,Y 463.75,Z 521.181,A -85,B 0,C 180,E1 -8049.386,E2 -8049.386} C_VEL
LIN {X 0,Y 463.533,Z 516.499,A -85,B 0,C 180,E1 -8050.704,E2 -8050.704} C_VEL
LIN {X 0,Y 462.075,Z 508.766,A -85,B 0,C 180,E1 -8053.192,E2 -8053.192} C_VEL
LIN {X 0,Y 460.88,Z 502.951,A -85,B 0,C 180,E1 -8055.456,E2 -8055.456} C_VEL
LIN {X 0,Y 460.534,Z 501.434,A -85,B 0,C 180,E1 -8056.212,E2 -8056.212} C_VEL
LIN {X 0,Y 460.535,Z 501.434,A -85,B 0,C 180,E1 -8058.99,E2 -8058.99} C_VEL
LIN {X 0,Y 460.528,Z 501.434,A -85,B 0,C 180,E1 -8061.268,E2 -8061.268} C_VEL
LIN {X 0,Y 460.514,Z 501.436,A -85,B 0,C 180,E1 -8064.555,E2 -8064.555} C_VEL
LIN {X 0,Y 460.533,Z 501.433,A -85,B 0,C 180,E1 -8067.716,E2 -8067.716} C_VEL
LIN {X 0,Y 460.541,Z 501.432,A -85,B 0,C 180,E1 -8070.77,E2 -8070.77} C_VEL
LIN {X 0,Y 460.569,Z 501.43,A -85,B 0,C 180,E1 -8073.812,E2 -8073.812} C_VEL
LIN {X 0,Y 460.577,Z 501.429,A -85,B 0,C 180,E1 -8073.874,E2 -8073.874} C_VEL
LIN {X 0,Y 461.624,Z 504.356,A -85,B 0,C 180,E1 -8074.018,E2 -8074.018} C_VEL
LIN {X 0,Y 467.195,Z 517.246,A -85,B 0,C 180,E1 -8074.751,E2 -8074.751} C_VEL
LIN {X 0,Y 469.716,Z 523.909,A -85,B 0,C 180,E1 -8075.144,E2 -8075.144} C_VEL
LIN {X 0,Y 469.025,Z 540.874,A -85,B 0,C 180,E1 -8075.86,E2 -8075.86} C_VEL
LIN {X 0,Y 468.145,Z 555.061,A -85,B 0,C 180,E1 -8076.615,E2 -8076.615} C_VEL
LIN {X 0,Y 467.194,Z 569.603,A -85,B 0,C 180,E1 -8077.56,E2 -8077.56} C_VEL
LIN {X 0,Y 466.183,Z 583.757,A -85,B 0,C 180,E1 -8078.673,E2 -8078.673} C_VEL
LIN {X 0,Y 465.126,Z 596.896,A -85,B 0,C 180,E1 -8079.895,E2 -8079.895} C_VEL
LIN {X 0,Y 464.116,Z 608.943,A -85,B 0,C 180,E1 -8081.23,E2 -8081.23} C_VEL
LIN {X 0,Y 463.217,Z 619.238,A -85,B 0,C 180,E1 -8082.564,E2 -8082.564} C_VEL
LIN {X 0,Y 462.345,Z 629.545,A -85,B 0,C 180,E1 -8084.121,E2 -8084.121} C_VEL
LIN {X 0,Y 461.536,Z 639.443,A -85,B 0,C 180,E1 -8085.899,E2 -8085.899} C_VEL
LIN {X 0,Y 461.001,Z 647.632,A -85,B 0,C 180,E1 -8087.677,E2 -8087.677} C_VEL
LIN {X 0,Y 460.419,Z 654.371,A -85,B 0,C 180,E1 -8089.446,E2 -8089.446} C_VEL
LIN {X 0,Y 460.138,Z 659.877,A -85,B 0,C 180,E1 -8091.215,E2 -8091.215} C_VEL
LIN {X 0,Y 459.954,Z 664.238,A -85,B 0,C 180,E1 -8092.979,E2 -8092.979} C_VEL
LIN {X 0,Y 459.801,Z 667.517,A -85,B 0,C 180,E1 -8094.738,E2 -8094.738} C_VEL
LIN {X 0,Y 459.75,Z 669.855,A -85,B 0,C 180,E1 -8096.495,E2 -8096.495} C_VEL
LIN {X 0,Y 459.657,Z 671.185,A -85,B 0,C 180,E1 -8098.248,E2 -8098.248} C_VEL
LIN {X 0,Y 459.581,Z 671.652,A -85,B 0,C 180,E1 -8100,E2 -8100} C_VEL
LIN {X 0,Y 459.647,Z 671.121,A -85,B 0,C 180,E1 -8101.753,E2 -8101.753} C_VEL
LIN {X 0,Y 459.748,Z 669.71,A -85,B 0,C 180,E1 -8103.506,E2 -8103.506} C_VEL
LIN {X 0,Y 459.74,Z 667.308,A -85,B 0,C 180,E1 -8105.263,E2 -8105.263} C_VEL
LIN {X 0,Y 459.902,Z 663.955,A -85,B 0,C 180,E1 -8107.023,E2 -8107.023} C_VEL
LIN {X 0,Y 460.131,Z 658.243,A -85,B 0,C 180,E1 -8109.229,E2 -8109.229} C_VEL
LIN {X 0,Y 460.408,Z 652.33,A -85,B 0,C 180,E1 -8111,E2 -8111} C_VEL
LIN {X 0,Y 460.902,Z 645.902,A -85,B 0,C 180,E1 -8112.605,E2 -8112.605} C_VEL
LIN {X 0,Y 461.432,Z 637.706,A -85,B 0,C 180,E1 -8114.33,E2 -8114.33} C_VEL
LIN {X 0,Y 462.285,Z 627.656,A -85,B 0,C 180,E1 -8116.09,E2 -8116.09} C_VEL
LIN {X 0,Y 463.104,Z 617.012,A -85,B 0,C 180,E1 -8117.669,E2 -8117.669} C_VEL
LIN {X 0,Y 464.161,Z 604.592,A -85,B 0,C 180,E1 -8119.228,E2 -8119.228} C_VEL
LIN {X 0,Y 465.289,Z 591.44,A -85,B 0,C 180,E1 -8120.62,E2 -8120.62} C_VEL
LIN {X 0,Y 466.363,Z 578.482,A -85,B 0,C 180,E1 -8121.784,E2 -8121.784} C_VEL
LIN {X 0,Y 467.368,Z 565.217,A -85,B 0,C 180,E1 -8122.782,E2 -8122.782} C_VEL
LIN {X 0,Y 468.408,Z 549.658,A -85,B 0,C 180,E1 -8123.759,E2 -8123.759} C_VEL
LIN {X 0,Y 469.399,Z 532.756,A -85,B 0,C 180,E1 -8124.603,E2 -8124.603} C_VEL
LIN {X 0,Y 469.681,Z 523.645,A -85,B 0,C 180,E1 -8124.982,E2 -8124.982} C_VEL
LIN {X 0,Y 463.071,Z 507.609,A -85,B 0,C 180,E1 -8125.918,E2 -8125.918} C_VEL
LIN {X 0,Y 460.625,Z 501.738,A -85,B 0,C 180,E1 -8126.229,E2 -8126.229} C_VEL
LIN {X 0,Y 460.582,Z 501.425,A -85,B 0,C 180,E1 -8126.265,E2 -8126.265} C_VEL
LIN {X 0,Y 460.544,Z 501.432,A -85,B 0,C 180,E1 -8129.231,E2 -8129.231} C_VEL
LIN {X 0,Y 460.536,Z 501.432,A -85,B 0,C 180,E1 -8132.285,E2 -8132.285} C_VEL
LIN {X 0,Y 460.518,Z 501.433,A -85,B 0,C 180,E1 -8135.445,E2 -8135.445} C_VEL
LIN {X 0,Y 460.55,Z 501.433,A -85,B 0,C 180,E1 -8138.898,E2 -8138.898} C_VEL
LIN {X 0,Y 460.528,Z 501.433,A -85,B 0,C 180,E1 -8142.181,E2 -8142.181} C_VEL
LIN {X 0,Y 460.519,Z 501.433,A -85,B 0,C 180,E1 -8145.411,E2 -8145.411} C_VEL
LIN {X 0,Y 460.538,Z 501.431,A -85,B 0,C 180,E1 -8148.397,E2 -8148.397} C_VEL
LIN {X 0,Y 460.532,Z 501.432,A -85,B 0,C 180,E1 -8151.267,E2 -8151.267} C_VEL
LIN {X 0,Y 460.516,Z 501.439,A -85,B 0,C 180,E1 -8154.554,E2 -8154.554} C_VEL
LIN {X 0,Y 460.537,Z 501.437,A -85,B 0,C 180,E1 -8157.715,E2 -8157.715} C_VEL
LIN {X 0,Y 460.545,Z 501.434,A -85,B 0,C 180,E1 -8160.769,E2 -8160.769} C_VEL
LIN {X 0,Y 460.594,Z 501.427,A -85,B 0,C 180,E1 -8163.736,E2 -8163.736} C_VEL
LIN {X 0,Y 460.674,Z 501.587,A -85,B 0,C 180,E1 -8164.711,E2 -8164.711} C_VEL
LIN {X 0,Y 460.814,Z 505.034,A -85,B 0,C 180,E1 -8166.638,E2 -8166.638} C_VEL
LIN {X 0,Y 460.756,Z 510.023,A -85,B 0,C 180,E1 -8169.462,E2 -8169.462} C_VEL
LIN {X 0,Y 460.732,Z 510.99,A -85,B 0,C 180,E1 -8170.019,E2 -8170.019} C_VEL
LIN {X 0,Y 460.062,Z 512.327,A -85,B 0,C 180,E1 -8170.729,E2 -8170.729} C_VEL
LIN {X 0,Y 457.182,Z 514.751,A -85,B 0,C 180,E1 -8171.875,E2 -8171.875} C_VEL
LIN {X 0,Y 454.754,Z 516.699,A -85,B 0,C 180,E1 -8172.798,E2 -8172.798} C_VEL
LIN {X 0,Y 453.728,Z 518.084,A -85,B 0,C 180,E1 -8173.516,E2 -8173.516} C_VEL
LIN {X 0,Y 453.654,Z 518.502,A -85,B 0,C 180,E1 -8173.76,E2 -8173.76} C_VEL
LIN {X 0,Y 453.542,Z 523.207,A -85,B 0,C 180,E1 -8176.559,E2 -8176.559} C_VEL
LIN {X 0,Y 453.573,Z 525.516,A -85,B 0,C 180,E1 -8177.933,E2 -8177.933} C_VEL
LIN {X 0,Y 455.364,Z 530.617,A -85,B 0,C 180,E1 -8178.135,E2 -8178.135} C_VEL
LIN {X 0,Y 461.402,Z 546.504,A -85,B 0,C 180,E1 -8178.877,E2 -8178.877} C_VEL
LIN {X 0,Y 464.167,Z 555.72,A -85,B 0,C 180,E1 -8179.338,E2 -8179.338} C_VEL
LIN {X 0,Y 463.402,Z 572.038,A -85,B 0,C 180,E1 -8179.959,E2 -8179.959} C_VEL
LIN {X 0,Y 462.492,Z 587.202,A -85,B 0,C 180,E1 -8180.708,E2 -8180.708} C_VEL
LIN {X 0,Y 461.312,Z 602.881,A -85,B 0,C 180,E1 -8181.677,E2 -8181.677} C_VEL
LIN {X 0,Y 460.023,Z 618.423,A -85,B 0,C 180,E1 -8182.869,E2 -8182.869} C_VEL
LIN {X 0,Y 458.825,Z 631.355,A -85,B 0,C 180,E1 -8184.065,E2 -8184.065} C_VEL
LIN {X 0,Y 457.635,Z 643.448,A -85,B 0,C 180,E1 -8185.375,E2 -8185.375} C_VEL
LIN {X 0,Y 456.468,Z 655.498,A -85,B 0,C 180,E1 -8186.91,E2 -8186.91} C_VEL
LIN {X 0,Y 455.469,Z 665.803,A -85,B 0,C 180,E1 -8188.452,E2 -8188.452} C_VEL
LIN {X 0,Y 454.483,Z 675.784,A -85,B 0,C 180,E1 -8190.221,E2 -8190.221} C_VEL
LIN {X 0,Y 453.91,Z 683.216,A -85,B 0,C 180,E1 -8191.774,E2 -8191.774} C_VEL
LIN {X 0,Y 453.325,Z 690.488,A -85,B 0,C 180,E1 -8193.554,E2 -8193.554} C_VEL
LIN {X 0,Y 452.922,Z 697.785,A -85,B 0,C 180,E1 -8195.788,E2 -8195.788} C_VEL
LIN {X 0,Y 452.685,Z 703.366,A -85,B 0,C 180,E1 -8198.031,E2 -8198.031} C_VEL
LIN {X 0,Y 452.451,Z 706.639,A -85,B 0,C 180,E1 -8199.837,E2 -8199.837} C_VEL
LIN {X 0,Y 452.492,Z 709.188,A -85,B 0,C 180,E1 -8201.9,E2 -8201.9} C_VEL
LIN {X 0,Y 452.337,Z 710.292,A -85,B 0,C 180,E1 -8203.476,E2 -8203.476} C_VEL
LIN {X 0,Y 452.359,Z 710.61,A -85,B 0,C 180,E1 -8205.579,E2 -8205.579} C_VEL
LIN {X 0,Y 452.344,Z 710.019,A -85,B 0,C 180,E1 -8207.168,E2 -8207.168} C_VEL
LIN {X 0,Y 452.377,Z 708.329,A -85,B 0,C 180,E1 -8209.04,E2 -8209.04} C_VEL
LIN {X 0,Y 452.538,Z 705.615,A -85,B 0,C 180,E1 -8210.927,E2 -8210.927} C_VEL
LIN {X 0,Y 452.712,Z 701.656,A -85,B 0,C 180,E1 -8212.835,E2 -8212.835} C_VEL
LIN {X 0,Y 453.007,Z 696.469,A -85,B 0,C 180,E1 -8214.763,E2 -8214.763} C_VEL
LIN {X 0,Y 453.437,Z 689.913,A -85,B 0,C 180,E1 -8216.709,E2 -8216.709} C_VEL
LIN {X 0,Y 454.027,Z 681.774,A -85,B 0,C 180,E1 -8218.675,E2 -8218.675} C_VEL
LIN {X 0,Y 454.757,Z 673.673,A -85,B 0,C 180,E1 -8220.294,E2 -8220.294} C_VEL
LIN {X 0,Y 455.648,Z 663.878,A -85,B 0,C 180,E1 -8221.969,E2 -8221.969} C_VEL
LIN {X 0,Y 456.805,Z 652.364,A -85,B 0,C 180,E1 -8223.631,E2 -8223.631} C_VEL
LIN {X 0,Y 457.989,Z 640.113,A -85,B 0,C 180,E1 -8225.13,E2 -8225.13} C_VEL
LIN {X 0,Y 459.307,Z 626.809,A -85,B 0,C 180,E1 -8226.499,E2 -8226.499} C_VEL
LIN {X 0,Y 460.6,Z 612.22,A -85,B 0,C 180,E1 -8227.75,E2 -8227.75} C_VEL
LIN {X 0,Y 461.757,Z 597.714,A -85,B 0,C 180,E1 -8228.777,E2 -8228.777} C_VEL
LIN {X 0,Y 462.797,Z 583.055,A -85,B 0,C 180,E1 -8229.627,E2 -8229.627} C_VEL
LIN {X 0,Y 463.699,Z 567.45,A -85,B 0,C 180,E1 -8230.35,E2 -8230.35} C_VEL
LIN {X 0,Y 464.128,Z 555.504,A -85,B 0,C 180,E1 -8230.789,E2 -8230.789} C_VEL
LIN {X 0,Y 461.121,Z 545.649,A -85,B 0,C 180,E1 -8231.291,E2 -8231.291} C_VEL
LIN {X 0,Y 454.75,Z 529.238,A -85,B 0,C 180,E1 -8232.082,E2 -8232.082} C_VEL
LIN {X 0,Y 453.637,Z 526.633,A -85,B 0,C 180,E1 -8232.205,E2 -8232.205} C_VEL
LIN {X 0,Y 453.514,Z 525.925,A -85,B 0,C 180,E1 -8232.243,E2 -8232.243} C_VEL
LIN {X 0,Y 453.653,Z 520.054,A -85,B 0,C 180,E1 -8235.801,E2 -8235.801} C_VEL
LIN {X 0,Y 453.79,Z 515.974,A -85,B 0,C 180,E1 -8238.244,E2 -8238.244} C_VEL
LIN {X 0,Y 453.833,Z 511.796,A -85,B 0,C 180,E1 -8240.739,E2 -8240.739} C_VEL
LIN {X 0,Y 453.954,Z 506.194,A -85,B 0,C 180,E1 -8243.963,E2 -8243.963} C_VEL
LIN {X 0,Y 453.531,Z 502.308,A -85,B 0,C 180,E1 -8246.23,E2 -8246.23} C_VEL
LIN {X 0,Y 453.475,Z 502.315,A -85,B 0,C 180,E1 -8249.24,E2 -8249.24} C_VEL
LIN {X 0,Y 453.536,Z 502.306,A -85,B 0,C 180,E1 -8252.297,E2 -8252.297} C_VEL
LIN {X 0,Y 453.517,Z 502.308,A -85,B 0,C 180,E1 -8255.265,E2 -8255.265} C_VEL
LIN {X 0,Y 453.473,Z 502.313,A -85,B 0,C 180,E1 -8258.413,E2 -8258.413} C_VEL
LIN {X 0,Y 453.513,Z 502.305,A -85,B 0,C 180,E1 -8261.008,E2 -8261.008} C_VEL
LIN {X 0,Y 453.558,Z 502.298,A -85,B 0,C 180,E1 -8263.879,E2 -8263.879} C_VEL
LIN {X 0,Y 453.591,Z 502.298,A -85,B 0,C 180,E1 -8267.472,E2 -8267.472} C_VEL
LIN {X 0,Y 453.583,Z 502.298,A -85,B 0,C 180,E1 -8271.086,E2 -8271.086} C_VEL
LIN {X 0,Y 453.674,Z 502.289,A -85,B 0,C 180,E1 -8273.774,E2 -8273.774} C_VEL
LIN {X 0,Y 453.757,Z 502.276,A -85,B 0,C 180,E1 -8277.336,E2 -8277.336} C_VEL
LIN {X 0,Y 453.813,Z 502.269,A -85,B 0,C 180,E1 -8280,E2 -8280} C_VEL
LIN {X 0,Y 453.757,Z 502.274,A -85,B 0,C 180,E1 -8282.663,E2 -8282.663} C_VEL
LIN {X 0,Y 453.666,Z 502.285,A -85,B 0,C 180,E1 -8286.225,E2 -8286.225} C_VEL
LIN {X 0,Y 453.582,Z 502.292,A -85,B 0,C 180,E1 -8288.913,E2 -8288.913} C_VEL
LIN {X 0,Y 453.59,Z 502.29,A -85,B 0,C 180,E1 -8292.551,E2 -8292.551} C_VEL
LIN {X 0,Y 453.533,Z 502.294,A -85,B 0,C 180,E1 -8296.196,E2 -8296.196} C_VEL
LIN {X 0,Y 453.509,Z 502.295,A -85,B 0,C 180,E1 -8299.041,E2 -8299.041} C_VEL
LIN {X 0,Y 453.49,Z 502.309,A -85,B 0,C 180,E1 -8301.835,E2 -8301.835} C_VEL
LIN {X 0,Y 453.514,Z 502.281,A -85,B 0,C 180,E1 -8304.734,E2 -8304.734} C_VEL
LIN {X 0,Y 453.527,Z 502.307,A -85,B 0,C 180,E1 -8307.962,E2 -8307.962} C_VEL
LIN {X 0,Y 453.472,Z 502.313,A -85,B 0,C 180,E1 -8310.759,E2 -8310.759} C_VEL
LIN {X 0,Y 453.467,Z 502.311,A -85,B 0,C 180,E1 -8313.913,E2 -8313.913} C_VEL
LIN {X 0,Y 453.463,Z 502.313,A -85,B 0,C 180,E1 -8317.188,E2 -8317.188} C_VEL
LIN {X 0,Y 453.527,Z 502.304,A -85,B 0,C 180,E1 -8319.445,E2 -8319.445} C_VEL
LIN {X 0,Y 453.524,Z 502.447,A -85,B 0,C 180,E1 -8321.711,E2 -8321.711} C_VEL
LIN {X 0,Y 455.493,Z 511.368,A -85,B 0,C 180,E1 -8324.787,E2 -8324.787} C_VEL
LIN {X 0,Y 457.303,Z 519.693,A -85,B 0,C 180,E1 -8327.534,E2 -8327.534} C_VEL
LIN {X 0,Y 458.27,Z 525.409,A -85,B 0,C 180,E1 -8329.336,E2 -8329.336} C_VEL
LIN {X 0,Y 458.057,Z 531.203,A -85,B 0,C 180,E1 -8331.021,E2 -8331.021} C_VEL
LIN {X 0,Y 457.337,Z 542.741,A -85,B 0,C 180,E1 -8334.273,E2 -8334.273} C_VEL
LIN {X 0,Y 456.652,Z 554.309,A -85,B 0,C 180,E1 -8337.409,E2 -8337.409} C_VEL
LIN {X 0,Y 455.928,Z 567.859,A -85,B 0,C 180,E1 -8340.952,E2 -8340.952} C_VEL
LIN {X 0,Y 455.552,Z 575.503,A -85,B 0,C 180,E1 -8342.887,E2 -8342.887} C_VEL
LIN {X 0,Y 460.947,Z 595.021,A -85,B 0,C 180,E1 -8343.605,E2 -8343.605} C_VEL
LIN {X 0,Y 464.085,Z 607.47,A -85,B 0,C 180,E1 -8344.148,E2 -8344.148} C_VEL
LIN {X 0,Y 463.348,Z 623.576,A -85,B 0,C 180,E1 -8344.722,E2 -8344.722} C_VEL
LIN {X 0,Y 462.317,Z 639.713,A -85,B 0,C 180,E1 -8345.47,E2 -8345.47} C_VEL
LIN {X 0,Y 461.067,Z 656.191,A -85,B 0,C 180,E1 -8346.44,E2 -8346.44} C_VEL
LIN {X 0,Y 459.83,Z 671.308,A -85,B 0,C 180,E1 -8347.538,E2 -8347.538} C_VEL
LIN {X 0,Y 458.599,Z 685.521,A -85,B 0,C 180,E1 -8348.775,E2 -8348.775} C_VEL
LIN {X 0,Y 457.459,Z 698.063,A -85,B 0,C 180,E1 -8350.057,E2 -8350.057} C_VEL
LIN {X 0,Y 456.272,Z 710.899,A -85,B 0,C 180,E1 -8351.594,E2 -8351.594} C_VEL
LIN {X 0,Y 455.294,Z 721.697,A -85,B 0,C 180,E1 -8353.144,E2 -8353.144} C_VEL
LIN {X 0,Y 454.467,Z 731.211,A -85,B 0,C 180,E1 -8354.759,E2 -8354.759} C_VEL
LIN {X 0,Y 453.735,Z 740.272,A -85,B 0,C 180,E1 -8356.566,E2 -8356.566} C_VEL
LIN {X 0,Y 453.26,Z 747.858,A -85,B 0,C 180,E1 -8358.372,E2 -8358.372} C_VEL
LIN {X 0,Y 452.79,Z 755.467,A -85,B 0,C 180,E1 -8360.621,E2 -8360.621} C_VEL
LIN {X 0,Y 452.644,Z 761.252,A -85,B 0,C 180,E1 -8362.866,E2 -8362.866} C_VEL
LIN {X 0,Y 452.499,Z 764.635,A -85,B 0,C 180,E1 -8364.654,E2 -8364.654} C_VEL
LIN {X 0,Y 452.431,Z 767.092,A -85,B 0,C 180,E1 -8366.439,E2 -8366.439} C_VEL
LIN {X 0,Y 452.427,Z 768.478,A -85,B 0,C 180,E1 -8368.221,E2 -8368.221} C_VEL
LIN {X 0,Y 452.377,Z 769,A -85,B 0,C 180,E1 -8370.001,E2 -8370.001} C_VEL
LIN {X 0,Y 452.427,Z 768.477,A -85,B 0,C 180,E1 -8371.781,E2 -8371.781} C_VEL
LIN {X 0,Y 452.431,Z 767.088,A -85,B 0,C 180,E1 -8373.563,E2 -8373.563} C_VEL
LIN {X 0,Y 452.5,Z 764.631,A -85,B 0,C 180,E1 -8375.348,E2 -8375.348} C_VEL
LIN {X 0,Y 452.645,Z 761.251,A -85,B 0,C 180,E1 -8377.136,E2 -8377.136} C_VEL
LIN {X 0,Y 452.791,Z 755.465,A -85,B 0,C 180,E1 -8379.381,E2 -8379.381} C_VEL
LIN {X 0,Y 453.24,Z 747.852,A -85,B 0,C 180,E1 -8381.63,E2 -8381.63} C_VEL
LIN {X 0,Y 453.824,Z 739.254,A -85,B 0,C 180,E1 -8383.661,E2 -8383.661} C_VEL
LIN {X 0,Y 454.618,Z 729.97,A -85,B 0,C 180,E1 -8385.467,E2 -8385.467} C_VEL
LIN {X 0,Y 455.441,Z 720.414,A -85,B 0,C 180,E1 -8387.05,E2 -8387.05} C_VEL
LIN {X 0,Y 456.279,Z 710.882,A -85,B 0,C 180,E1 -8388.407,E2 -8388.407} C_VEL
LIN {X 0,Y 457.263,Z 699.495,A -85,B 0,C 180,E1 -8389.764,E2 -8389.764} C_VEL
LIN {X 0,Y 458.448,Z 686.271,A -85,B 0,C 180,E1 -8391.117,E2 -8391.117} C_VEL
LIN {X 0,Y 459.665,Z 671.975,A -85,B 0,C 180,E1 -8392.354,E2 -8392.354} C_VEL
LIN {X 0,Y 460.812,Z 658.113,A -85,B 0,C 180,E1 -8393.362,E2 -8393.362} C_VEL
LIN {X 0,Y 461.776,Z 644.615,A -85,B 0,C 180,E1 -8394.188,E2 -8394.188} C_VEL
LIN {X 0,Y 462.842,Z 628.947,A -85,B 0,C 180,E1 -8394.982,E2 -8394.982} C_VEL
LIN {X 0,Y 463.583,Z 615.449,A -85,B 0,C 180,E1 -8395.522,E2 -8395.522} C_VEL
LIN {X 0,Y 463.842,Z 607.171,A -85,B 0,C 180,E1 -8395.805,E2 -8395.805} C_VEL
LIN {X 0,Y 459.516,Z 590.503,A -85,B 0,C 180,E1 -8396.527,E2 -8396.527} C_VEL
LIN {X 0,Y 456.905,Z 580.007,A -85,B 0,C 180,E1 -8396.913,E2 -8396.913} C_VEL
LIN {X 0,Y 455.28,Z 572.245,A -85,B 0,C 180,E1 -8397.195,E2 -8397.195} C_VEL
LIN {X 0,Y 455.684,Z 559.195,A -85,B 0,C 180,E1 -8400.268,E2 -8400.268} C_VEL
LIN {X 0,Y 456.047,Z 546.089,A -85,B 0,C 180,E1 -8403.423,E2 -8403.423} C_VEL
LIN {X 0,Y 456.406,Z 534.496,A -85,B 0,C 180,E1 -8406.313,E2 -8406.313} C_VEL
LIN {X 0,Y 456.81,Z 522.779,A -85,B 0,C 180,E1 -8409.414,E2 -8409.414} C_VEL
LIN {X 0,Y 456.709,Z 518.553,A -85,B 0,C 180,E1 -8410.629,E2 -8410.629} C_VEL
LIN {X 0,Y 455.514,Z 512.032,A -85,B 0,C 180,E1 -8412.756,E2 -8412.756} C_VEL
LIN {X 0,Y 454.493,Z 507.012,A -85,B 0,C 180,E1 -8414.658,E2 -8414.658} C_VEL
LIN {X 0,Y 453.466,Z 502.314,A -85,B 0,C 180,E1 -8416.894,E2 -8416.894} C_VEL
LIN {X 0,Y 453.496,Z 502.31,A -85,B 0,C 180,E1 -8419.409,E2 -8419.409} C_VEL
LIN {X 0,Y 453.474,Z 502.313,A -85,B 0,C 180,E1 -8422.224,E2 -8422.224} C_VEL
LIN {X 0,Y 453.49,Z 502.31,A -85,B 0,C 180,E1 -8425.223,E2 -8425.223} C_VEL
LIN {X 0,Y 453.467,Z 502.314,A -85,B 0,C 180,E1 -8428.475,E2 -8428.475} C_VEL
LIN {X 0,Y 453.539,Z 502.306,A -85,B 0,C 180,E1 -8432.04,E2 -8432.04} C_VEL
LIN {X 0,Y 453.538,Z 502.304,A -85,B 0,C 180,E1 -8433.414,E2 -8433.414} C_VEL
LIN {X 0,Y 454.468,Z 505.043,A -85,B 0,C 180,E1 -8433.558,E2 -8433.558} C_VEL
LIN {X 0,Y 459.676,Z 516.468,A -85,B 0,C 180,E1 -8434.253,E2 -8434.253} C_VEL
LIN {X 0,Y 463.303,Z 526.189,A -85,B 0,C 180,E1 -8434.846,E2 -8434.846} C_VEL
LIN {X 0,Y 462.554,Z 541.715,A -85,B 0,C 180,E1 -8435.518,E2 -8435.518} C_VEL
LIN {X 0,Y 461.637,Z 556.037,A -85,B 0,C 180,E1 -8436.295,E2 -8436.295} C_VEL
LIN {X 0,Y 460.646,Z 570.137,A -85,B 0,C 180,E1 -8437.224,E2 -8437.224} C_VEL
LIN {X 0,Y 459.59,Z 584.386,A -85,B 0,C 180,E1 -8438.352,E2 -8438.352} C_VEL
LIN {X 0,Y 458.469,Z 597.523,A -85,B 0,C 180,E1 -8439.59,E2 -8439.59} C_VEL
LIN {X 0,Y 457.414,Z 609.557,A -85,B 0,C 180,E1 -8440.944,E2 -8440.944} C_VEL
LIN {X 0,Y 456.444,Z 619.927,A -85,B 0,C 180,E1 -8442.297,E2 -8442.297} C_VEL
LIN {X 0,Y 455.536,Z 630.285,A -85,B 0,C 180,E1 -8443.877,E2 -8443.877} C_VEL
LIN {X 0,Y 454.669,Z 640.21,A -85,B 0,C 180,E1 -8445.682,E2 -8445.682} C_VEL
LIN {X 0,Y 454.088,Z 648.407,A -85,B 0,C 180,E1 -8447.486,E2 -8447.486} C_VEL
LIN {X 0,Y 453.474,Z 655.176,A -85,B 0,C 180,E1 -8449.282,E2 -8449.282} C_VEL
LIN {X 0,Y 453.158,Z 660.702,A -85,B 0,C 180,E1 -8451.078,E2 -8451.078} C_VEL
LIN {X 0,Y 452.946,Z 665.063,A -85,B 0,C 180,E1 -8452.87,E2 -8452.87} C_VEL
LIN {X 0,Y 452.788,Z 668.346,A -85,B 0,C 180,E1 -8454.657,E2 -8454.657} C_VEL
LIN {X 0,Y 452.713,Z 670.679,A -85,B 0,C 180,E1 -8456.44,E2 -8456.44} C_VEL
LIN {X 0,Y 452.605,Z 671.998,A -85,B 0,C 180,E1 -8458.221,E2 -8458.221} C_VEL
LIN {X 0,Y 452.528,Z 672.458,A -85,B 0,C 180,E1 -8460,E2 -8460} C_VEL
LIN {X 0,Y 452.591,Z 671.898,A -85,B 0,C 180,E1 -8461.78,E2 -8461.78} C_VEL
LIN {X 0,Y 452.71,Z 670.48,A -85,B 0,C 180,E1 -8463.561,E2 -8463.561} C_VEL
LIN {X 0,Y 452.71,Z 668.036,A -85,B 0,C 180,E1 -8465.345,E2 -8465.345} C_VEL
LIN {X 0,Y 452.889,Z 664.662,A -85,B 0,C 180,E1 -8467.132,E2 -8467.132} C_VEL
LIN {X 0,Y 453.12,Z 658.9,A -85,B 0,C 180,E1 -8469.373,E2 -8469.373} C_VEL
LIN {X 0,Y 453.446,Z 652.946,A -85,B 0,C 180,E1 -8471.171,E2 -8471.171} C_VEL
LIN {X 0,Y 453.961,Z 645.719,A -85,B 0,C 180,E1 -8472.972,E2 -8472.972} C_VEL
LIN {X 0,Y 454.621,Z 637.032,A -85,B 0,C 180,E1 -8474.778,E2 -8474.778} C_VEL
LIN {X 0,Y 455.512,Z 627.066,A -85,B 0,C 180,E1 -8476.517,E2 -8476.517} C_VEL
LIN {X 0,Y 456.462,Z 615.804,A -85,B 0,C 180,E1 -8478.167,E2 -8478.167} C_VEL
LIN {X 0,Y 457.442,Z 604.936,A -85,B 0,C 180,E1 -8479.522,E2 -8479.522} C_VEL
LIN {X 0,Y 458.598,Z 591.976,A -85,B 0,C 180,E1 -8480.909,E2 -8480.909} C_VEL
LIN {X 0,Y 459.752,Z 578.688,A -85,B 0,C 180,E1 -8482.113,E2 -8482.113} C_VEL
LIN {X 0,Y 460.82,Z 565.37,A -85,B 0,C 180,E1 -8483.124,E2 -8483.124} C_VEL
LIN {X 0,Y 461.812,Z 550.653,A -85,B 0,C 180,E1 -8484.062,E2 -8484.062} C_VEL
LIN {X 0,Y 462.827,Z 534.918,A -85,B 0,C 180,E1 -8484.87,E2 -8484.87} C_VEL
LIN {X 0,Y 463.17,Z 525.857,A -85,B 0,C 180,E1 -8485.261,E2 -8485.261} C_VEL
LIN {X 0,Y 457.334,Z 511.367,A -85,B 0,C 180,E1 -8486.145,E2 -8486.145} C_VEL
LIN {X 0,Y 453.608,Z 502.784,A -85,B 0,C 180,E1 -8486.62,E2 -8486.62} C_VEL
LIN {X 0,Y 453.531,Z 502.305,A -85,B 0,C 180,E1 -8486.656,E2 -8486.656} C_VEL
LIN {X 0,Y 453.477,Z 502.312,A -85,B 0,C 180,E1 -8489.785,E2 -8489.785} C_VEL
LIN {X 0,Y 453.495,Z 502.311,A -85,B 0,C 180,E1 -8493.189,E2 -8493.189} C_VEL
LIN {X 0,Y 453.46,Z 502.314,A -85,B 0,C 180,E1 -8496.3,E2 -8496.3} C_VEL
LIN {X 0,Y 453.495,Z 502.309,A -85,B 0,C 180,E1 -8499.45,E2 -8499.45} C_VEL
LIN {X 0,Y 453.481,Z 502.313,A -85,B 0,C 180,E1 -8501.935,E2 -8501.935} C_VEL
LIN {X 0,Y 453.489,Z 502.309,A -85,B 0,C 180,E1 -8505.471,E2 -8505.471} C_VEL
LIN {X 0,Y 453.485,Z 502.309,A -85,B 0,C 180,E1 -8508.209,E2 -8508.209} C_VEL
LIN {X 0,Y 453.521,Z 502.306,A -85,B 0,C 180,E1 -8510.79,E2 -8510.79} C_VEL
LIN {X 0,Y 453.46,Z 502.315,A -85,B 0,C 180,E1 -8513.917,E2 -8513.917} C_VEL
LIN {X 0,Y 453.489,Z 502.313,A -85,B 0,C 180,E1 -8517.151,E2 -8517.151} C_VEL
LIN {X 0,Y 453.481,Z 502.315,A -85,B 0,C 180,E1 -8520.268,E2 -8520.268} C_VEL
LIN {X 0,Y 453.541,Z 502.306,A -85,B 0,C 180,E1 -8523.295,E2 -8523.295} C_VEL
LIN {X 0,Y 453.64,Z 502.441,A -85,B 0,C 180,E1 -8524.537,E2 -8524.537} C_VEL
LIN {X 0,Y 453.864,Z 505.513,A -85,B 0,C 180,E1 -8526.258,E2 -8526.258} C_VEL
LIN {X 0,Y 453.737,Z 510.561,A -85,B 0,C 180,E1 -8529.129,E2 -8529.129} C_VEL
LIN {X 0,Y 453.7,Z 515.426,A -85,B 0,C 180,E1 -8531.952,E2 -8531.952} C_VEL
LIN {X 0,Y 453.654,Z 518.502,A -85,B 0,C 180,E1 -8533.76,E2 -8533.76} C_VEL
LIN {X 0,Y 452.982,Z 519.426,A -85,B 0,C 180,E1 -8534.24,E2 -8534.24} C_VEL
LIN {X 0,Y 450.105,Z 521.133,A -85,B 0,C 180,E1 -8534.982,E2 -8534.982} C_VEL
LIN {X 0,Y 447.211,Z 522.843,A -85,B 0,C 180,E1 -8535.733,E2 -8535.733} C_VEL
LIN {X 0,Y 446.532,Z 523.772,A -85,B 0,C 180,E1 -8536.223,E2 -8536.223} C_VEL
LIN {X 0,Y 446.561,Z 525.86,A -85,B 0,C 180,E1 -8537.485,E2 -8537.485} C_VEL
LIN {X 0,Y 451.923,Z 539.909,A -85,B 0,C 180,E1 -8538.115,E2 -8538.115} C_VEL
LIN {X 0,Y 456.919,Z 554.318,A -85,B 0,C 180,E1 -8538.844,E2 -8538.844} C_VEL
LIN {X 0,Y 457.786,Z 557.837,A -85,B 0,C 180,E1 -8539.021,E2 -8539.021} C_VEL
LIN {X 0,Y 456.924,Z 573.633,A -85,B 0,C 180,E1 -8539.643,E2 -8539.643} C_VEL
LIN {X 0,Y 455.855,Z 589.556,A -85,B 0,C 180,E1 -8540.459,E2 -8540.459} C_VEL
LIN {X 0,Y 454.777,Z 603.366,A -85,B 0,C 180,E1 -8541.333,E2 -8541.333} C_VEL
LIN {X 0,Y 453.427,Z 618.903,A -85,B 0,C 180,E1 -8542.541,E2 -8542.541} C_VEL
LIN {X 0,Y 452.152,Z 631.846,A -85,B 0,C 180,E1 -8543.753,E2 -8543.753} C_VEL
LIN {X 0,Y 450.934,Z 643.934,A -85,B 0,C 180,E1 -8545.082,E2 -8545.082} C_VEL
LIN {X 0,Y 449.683,Z 655.995,A -85,B 0,C 180,E1 -8546.639,E2 -8546.639} C_VEL
LIN {X 0,Y 448.633,Z 666.3,A -85,B 0,C 180,E1 -8548.204,E2 -8548.204} C_VEL
LIN {X 0,Y 447.584,Z 676.274,A -85,B 0,C 180,E1 -8549.999,E2 -8549.999} C_VEL
LIN {X 0,Y 446.872,Z 684.666,A -85,B 0,C 180,E1 -8551.802,E2 -8551.802} C_VEL
LIN {X 0,Y 446.276,Z 691.75,A -85,B 0,C 180,E1 -8553.611,E2 -8553.611} C_VEL
LIN {X 0,Y 445.946,Z 697.581,A -85,B 0,C 180,E1 -8555.425,E2 -8555.425} C_VEL
LIN {X 0,Y 445.703,Z 702.284,A -85,B 0,C 180,E1 -8557.246,E2 -8557.246} C_VEL
LIN {X 0,Y 445.461,Z 706.023,A -85,B 0,C 180,E1 -8559.076,E2 -8559.076} C_VEL
LIN {X 0,Y 445.417,Z 708.648,A -85,B 0,C 180,E1 -8560.913,E2 -8560.913} C_VEL
LIN {X 0,Y 445.309,Z 710.384,A -85,B 0,C 180,E1 -8562.764,E2 -8562.764} C_VEL
LIN {X 0,Y 445.273,Z 711.078,A -85,B 0,C 180,E1 -8564.627,E2 -8564.627} C_VEL
LIN {X 0,Y 445.242,Z 710.824,A -85,B 0,C 180,E1 -8566.505,E2 -8566.505} C_VEL
LIN {X 0,Y 445.303,Z 709.539,A -85,B 0,C 180,E1 -8568.399,E2 -8568.399} C_VEL
LIN {X 0,Y 445.386,Z 707.172,A -85,B 0,C 180,E1 -8570.312,E2 -8570.312} C_VEL
LIN {X 0,Y 445.642,Z 703.733,A -85,B 0,C 180,E1 -8572.239,E2 -8572.239} C_VEL
LIN {X 0,Y 445.886,Z 699.004,A -85,B 0,C 180,E1 -8574.191,E2 -8574.191} C_VEL
LIN {X 0,Y 446.272,Z 692.943,A -85,B 0,C 180,E1 -8576.163,E2 -8576.163} C_VEL
LIN {X 0,Y 446.858,Z 685.395,A -85,B 0,C 180,E1 -8578.152,E2 -8578.152} C_VEL
LIN {X 0,Y 447.587,Z 677.418,A -85,B 0,C 180,E1 -8579.902,E2 -8579.902} C_VEL
LIN {X 0,Y 448.5,Z 667.83,A -85,B 0,C 180,E1 -8581.663,E2 -8581.663} C_VEL
LIN {X 0,Y 449.682,Z 656.407,A -85,B 0,C 180,E1 -8583.428,E2 -8583.428} C_VEL
LIN {X 0,Y 450.875,Z 644.769,A -85,B 0,C 180,E1 -8584.947,E2 -8584.947} C_VEL
LIN {X 0,Y 452.179,Z 632.223,A -85,B 0,C 180,E1 -8586.337,E2 -8586.337} C_VEL
LIN {X 0,Y 453.538,Z 619.167,A -85,B 0,C 180,E1 -8587.561,E2 -8587.561} C_VEL
LIN {X 0,Y 454.839,Z 604.152,A -85,B 0,C 180,E1 -8588.738,E2 -8588.738} C_VEL
LIN {X 0,Y 455.972,Z 589.412,A -85,B 0,C 180,E1 -8589.68,E2 -8589.68} C_VEL
LIN {X 0,Y 457.03,Z 573.906,A -85,B 0,C 180,E1 -8590.474,E2 -8590.474} C_VEL
LIN {X 0,Y 457.802,Z 557.345,A -85,B 0,C 180,E1 -8591.132,E2 -8591.132} C_VEL
LIN {X 0,Y 454.963,Z 548.036,A -85,B 0,C 180,E1 -8591.627,E2 -8591.627} C_VEL
LIN {X 0,Y 449.132,Z 532.858,A -85,B 0,C 180,E1 -8592.407,E2 -8592.407} C_VEL
LIN {X 0,Y 446.636,Z 526.945,A -85,B 0,C 180,E1 -8592.692,E2 -8592.692} C_VEL
LIN {X 0,Y 446.53,Z 526.318,A -85,B 0,C 180,E1 -8592.754,E2 -8592.754} C_VEL
LIN {X 0,Y 446.669,Z 520.682,A -85,B 0,C 180,E1 -8596.186,E2 -8596.186} C_VEL
LIN {X 0,Y 446.81,Z 516.011,A -85,B 0,C 180,E1 -8599.024,E2 -8599.024} C_VEL
LIN {X 0,Y 446.89,Z 510.718,A -85,B 0,C 180,E1 -8602.169,E2 -8602.169} C_VEL
LIN {X 0,Y 446.906,Z 506.046,A -85,B 0,C 180,E1 -8604.857,E2 -8604.857} C_VEL
LIN {X 0,Y 446.457,Z 503.19,A -85,B 0,C 180,E1 -8606.567,E2 -8606.567} C_VEL
LIN {X 0,Y 446.433,Z 503.192,A -85,B 0,C 180,E1 -8609.976,E2 -8609.976} C_VEL
LIN {X 0,Y 446.474,Z 503.184,A -85,B 0,C 180,E1 -8612.838,E2 -8612.838} C_VEL
LIN {X 0,Y 446.458,Z 503.188,A -85,B 0,C 180,E1 -8615.922,E2 -8615.922} C_VEL
LIN {X 0,Y 446.45,Z 503.187,A -85,B 0,C 180,E1 -8618.772,E2 -8618.772} C_VEL
LIN {X 0,Y 446.448,Z 503.187,A -85,B 0,C 180,E1 -8621.648,E2 -8621.648} C_VEL
LIN {X 0,Y 446.497,Z 503.182,A -85,B 0,C 180,E1 -8624.479,E2 -8624.479} C_VEL
LIN {X 0,Y 446.53,Z 503.178,A -85,B 0,C 180,E1 -8628.193,E2 -8628.193} C_VEL
LIN {X 0,Y 446.59,Z 503.164,A -85,B 0,C 180,E1 -8631.857,E2 -8631.857} C_VEL
LIN {X 0,Y 446.644,Z 503.16,A -85,B 0,C 180,E1 -8634.582,E2 -8634.582} C_VEL
LIN {X 0,Y 446.701,Z 503.155,A -85,B 0,C 180,E1 -8637.294,E2 -8637.294} C_VEL
LIN {X 0,Y 446.784,Z 503.145,A -85,B 0,C 180,E1 -8640,E2 -8640} C_VEL
LIN {X 0,Y 446.7,Z 503.153,A -85,B 0,C 180,E1 -8642.705,E2 -8642.705} C_VEL
LIN {X 0,Y 446.635,Z 503.162,A -85,B 0,C 180,E1 -8646.323,E2 -8646.323} C_VEL
LIN {X 0,Y 446.528,Z 503.171,A -85,B 0,C 180,E1 -8649.055,E2 -8649.055} C_VEL
LIN {X 0,Y 446.523,Z 503.171,A -85,B 0,C 180,E1 -8652.729,E2 -8652.729} C_VEL
LIN {X 0,Y 446.478,Z 503.167,A -85,B 0,C 180,E1 -8656.459,E2 -8656.459} C_VEL
LIN {X 0,Y 446.459,Z 503.175,A -85,B 0,C 180,E1 -8659.303,E2 -8659.303} C_VEL
LIN {X 0,Y 446.426,Z 503.188,A -85,B 0,C 180,E1 -8662.199,E2 -8662.199} C_VEL
LIN {X 0,Y 446.46,Z 503.162,A -85,B 0,C 180,E1 -8665.152,E2 -8665.152} C_VEL
LIN {X 0,Y 446.473,Z 503.184,A -85,B 0,C 180,E1 -8668.179,E2 -8668.179} C_VEL
LIN {X 0,Y 446.409,Z 503.191,A -85,B 0,C 180,E1 -8671.3,E2 -8671.3} C_VEL
LIN {X 0,Y 446.42,Z 503.19,A -85,B 0,C 180,E1 -8674.523,E2 -8674.523} C_VEL
LIN {X 0,Y 446.43,Z 503.187,A -85,B 0,C 180,E1 -8678.084,E2 -8678.084} C_VEL
LIN {X 0,Y 446.458,Z 503.185,A -85,B 0,C 180,E1 -8681.118,E2 -8681.118} C_VEL
LIN {X 0,Y 448.106,Z 510.654,A -85,B 0,C 180,E1 -8683.827,E2 -8683.827} C_VEL
LIN {X 0,Y 449.868,Z 518.803,A -85,B 0,C 180,E1 -8686.579,E2 -8686.579} C_VEL
LIN {X 0,Y 451.278,Z 525.615,A -85,B 0,C 180,E1 -8688.794,E2 -8688.794} C_VEL
LIN {X 0,Y 451.356,Z 530.703,A -85,B 0,C 180,E1 -8690.329,E2 -8690.329} C_VEL
LIN {X 0,Y 450.575,Z 542.285,A -85,B 0,C 180,E1 -8693.652,E2 -8693.652} C_VEL
LIN {X 0,Y 449.725,Z 555.346,A -85,B 0,C 180,E1 -8697.262,E2 -8697.262} C_VEL
LIN {X 0,Y 448.927,Z 569.259,A -85,B 0,C 180,E1 -8700.969,E2 -8700.969} C_VEL
LIN {X 0,Y 448.589,Z 574.734,A -85,B 0,C 180,E1 -8702.414,E2 -8702.414} C_VEL
LIN {X 0,Y 454.364,Z 596.055,A -85,B 0,C 180,E1 -8703.234,E2 -8703.234} C_VEL
LIN {X 0,Y 457.629,Z 609.131,A -85,B 0,C 180,E1 -8703.831,E2 -8703.831} C_VEL
LIN {X 0,Y 456.812,Z 624.149,A -85,B 0,C 180,E1 -8704.393,E2 -8704.393} C_VEL
LIN {X 0,Y 455.705,Z 640.013,A -85,B 0,C 180,E1 -8705.151,E2 -8705.151} C_VEL
LIN {X 0,Y 454.538,Z 654.923,A -85,B 0,C 180,E1 -8706.045,E2 -8706.045} C_VEL
LIN {X 0,Y 453.103,Z 670.552,A -85,B 0,C 180,E1 -8707.185,E2 -8707.185} C_VEL
LIN {X 0,Y 451.857,Z 684.768,A -85,B 0,C 180,E1 -8708.443,E2 -8708.443} C_VEL
LIN {X 0,Y 450.615,Z 697.485,A -85,B 0,C 180,E1 -8709.761,E2 -8709.761} C_VEL
LIN {X 0,Y 449.379,Z 710.155,A -85,B 0,C 180,E1 -8711.302,E2 -8711.302} C_VEL
LIN {X 0,Y 448.304,Z 721.927,A -85,B 0,C 180,E1 -8712.996,E2 -8712.996} C_VEL
LIN {X 0,Y 447.542,Z 730.942,A -85,B 0,C 180,E1 -8714.518,E2 -8714.518} C_VEL
LIN {X 0,Y 446.763,Z 740.255,A -85,B 0,C 180,E1 -8716.353,E2 -8716.353} C_VEL
LIN {X 0,Y 446.232,Z 747.858,A -85,B 0,C 180,E1 -8718.187,E2 -8718.187} C_VEL
LIN {X 0,Y 445.735,Z 755.467,A -85,B 0,C 180,E1 -8720.472,E2 -8720.472} C_VEL
LIN {X 0,Y 445.568,Z 761.252,A -85,B 0,C 180,E1 -8722.752,E2 -8722.752} C_VEL
LIN {X 0,Y 445.42,Z 764.635,A -85,B 0,C 180,E1 -8724.569,E2 -8724.569} C_VEL
LIN {X 0,Y 445.329,Z 767.092,A -85,B 0,C 180,E1 -8726.382,E2 -8726.382} C_VEL
LIN {X 0,Y 445.346,Z 768.478,A -85,B 0,C 180,E1 -8728.192,E2 -8728.192} C_VEL
LIN {X 0,Y 445.287,Z 769,A -85,B 0,C 180,E1 -8730.001,E2 -8730.001} C_VEL
LIN {X 0,Y 445.347,Z 768.476,A -85,B 0,C 180,E1 -8731.81,E2 -8731.81} C_VEL
LIN {X 0,Y 445.33,Z 767.088,A -85,B 0,C 180,E1 -8733.62,E2 -8733.62} C_VEL
LIN {X 0,Y 445.421,Z 764.631,A -85,B 0,C 180,E1 -8735.433,E2 -8735.433} C_VEL
LIN {X 0,Y 445.57,Z 761.251,A -85,B 0,C 180,E1 -8737.25,E2 -8737.25} C_VEL
LIN {X 0,Y 445.736,Z 755.465,A -85,B 0,C 180,E1 -8739.53,E2 -8739.53} C_VEL
LIN {X 0,Y 446.224,Z 747.852,A -85,B 0,C 180,E1 -8741.816,E2 -8741.816} C_VEL
LIN {X 0,Y 446.766,Z 740.246,A -85,B 0,C 180,E1 -8743.649,E2 -8743.649} C_VEL
LIN {X 0,Y 447.399,Z 732.158,A -85,B 0,C 180,E1 -8745.256,E2 -8745.256} C_VEL
LIN {X 0,Y 448.223,Z 722.69,A -85,B 0,C 180,E1 -8746.855,E2 -8746.855} C_VEL
LIN {X 0,Y 449.224,Z 711.42,A -85,B 0,C 180,E1 -8748.471,E2 -8748.471} C_VEL
LIN {X 0,Y 450.304,Z 699.241,A -85,B 0,C 180,E1 -8749.963,E2 -8749.963} C_VEL
LIN {X 0,Y 451.563,Z 686.133,A -85,B 0,C 180,E1 -8751.335,E2 -8751.335} C_VEL
LIN {X 0,Y 452.812,Z 671.994,A -85,B 0,C 180,E1 -8752.591,E2 -8752.591} C_VEL
LIN {X 0,Y 454.14,Z 656.662,A -85,B 0,C 180,E1 -8753.727,E2 -8753.727} C_VEL
LIN {X 0,Y 455.327,Z 640.8,A -85,B 0,C 180,E1 -8754.691,E2 -8754.691} C_VEL
LIN {X 0,Y 456.464,Z 624.749,A -85,B 0,C 180,E1 -8755.477,E2 -8755.477} C_VEL
LIN {X 0,Y 457.252,Z 608.579,A -85,B 0,C 180,E1 -8756.108,E2 -8756.108} C_VEL
LIN {X 0,Y 452.666,Z 590.531,A -85,B 0,C 180,E1 -8756.931,E2 -8756.931} C_VEL
LIN {X 0,Y 448.293,Z 571.084,A -85,B 0,C 180,E1 -8757.648,E2 -8757.648} C_VEL
LIN {X 0,Y 448.721,Z 558.012,A -85,B 0,C 180,E1 -8760.772,E2 -8760.772} C_VEL
LIN {X 0,Y 449.117,Z 545.083,A -85,B 0,C 180,E1 -8763.967,E2 -8763.967} C_VEL
LIN {X 0,Y 449.501,Z 534.113,A -85,B 0,C 180,E1 -8766.789,E2 -8766.789} C_VEL
LIN {X 0,Y 449.956,Z 522.247,A -85,B 0,C 180,E1 -8770.063,E2 -8770.063} C_VEL
LIN {X 0,Y 449.148,Z 516.469,A -85,B 0,C 180,E1 -8771.907,E2 -8771.907} C_VEL
LIN {X 0,Y 447.834,Z 509.703,A -85,B 0,C 180,E1 -8774.436,E2 -8774.436} C_VEL
LIN {X 0,Y 446.963,Z 505.603,A -85,B 0,C 180,E1 -8776.328,E2 -8776.328} C_VEL
LIN {X 0,Y 446.438,Z 503.189,A -85,B 0,C 180,E1 -8777.723,E2 -8777.723} C_VEL
LIN {X 0,Y 446.458,Z 503.187,A -85,B 0,C 180,E1 -8780.975,E2 -8780.975} C_VEL
LIN {X 0,Y 446.422,Z 503.192,A -85,B 0,C 180,E1 -8784.375,E2 -8784.375} C_VEL
LIN {X 0,Y 446.424,Z 503.191,A -85,B 0,C 180,E1 -8787.639,E2 -8787.639} C_VEL
LIN {X 0,Y 446.451,Z 503.187,A -85,B 0,C 180,E1 -8790.791,E2 -8790.791} C_VEL
LIN {X 0,Y 446.485,Z 503.214,A -85,B 0,C 180,E1 -8792.924,E2 -8792.924} C_VEL
LIN {X 0,Y 447.466,Z 506.037,A -85,B 0,C 180,E1 -8793.082,E2 -8793.082} C_VEL
LIN {X 0,Y 452.604,Z 516.785,A -85,B 0,C 180,E1 -8793.79,E2 -8793.79} C_VEL
LIN {X 0,Y 456.652,Z 527.534,A -85,B 0,C 180,E1 -8794.474,E2 -8794.474} C_VEL
LIN {X 0,Y 456.369,Z 537.671,A -85,B 0,C 180,E1 -8794.924,E2 -8794.924} C_VEL
LIN {X 0,Y 455.39,Z 553.729,A -85,B 0,C 180,E1 -8795.759,E2 -8795.759} C_VEL
LIN {X 0,Y 454.242,Z 569.324,A -85,B 0,C 180,E1 -8796.763,E2 -8796.763} C_VEL
LIN {X 0,Y 453.131,Z 583.778,A -85,B 0,C 180,E1 -8797.907,E2 -8797.907} C_VEL
LIN {X 0,Y 451.819,Z 598.199,A -85,B 0,C 180,E1 -8799.276,E2 -8799.276} C_VEL
LIN {X 0,Y 450.72,Z 610.288,A -85,B 0,C 180,E1 -8800.65,E2 -8800.65} C_VEL
LIN {X 0,Y 449.548,Z 622.245,A -85,B 0,C 180,E1 -8802.252,E2 -8802.252} C_VEL
LIN {X 0,Y 448.615,Z 632.343,A -85,B 0,C 180,E1 -8803.855,E2 -8803.855} C_VEL
LIN {X 0,Y 447.812,Z 640.997,A -85,B 0,C 180,E1 -8805.457,E2 -8805.457} C_VEL
LIN {X 0,Y 447.174,Z 649.208,A -85,B 0,C 180,E1 -8807.29,E2 -8807.29} C_VEL
LIN {X 0,Y 446.533,Z 655.991,A -85,B 0,C 180,E1 -8809.114,E2 -8809.114} C_VEL
LIN {X 0,Y 446.182,Z 661.528,A -85,B 0,C 180,E1 -8810.938,E2 -8810.938} C_VEL
LIN {X 0,Y 445.927,Z 665.893,A -85,B 0,C 180,E1 -8812.757,E2 -8812.757} C_VEL
LIN {X 0,Y 445.775,Z 669.178,A -85,B 0,C 180,E1 -8814.572,E2 -8814.572} C_VEL
LIN {X 0,Y 445.678,Z 671.506,A -85,B 0,C 180,E1 -8816.384,E2 -8816.384} C_VEL
LIN {X 0,Y 445.553,Z 672.814,A -85,B 0,C 180,E1 -8818.193,E2 -8818.193} C_VEL
LIN {X 0,Y 445.475,Z 673.265,A -85,B 0,C 180,E1 -8820,E2 -8820} C_VEL
LIN {X 0,Y 445.535,Z 672.678,A -85,B 0,C 180,E1 -8821.808,E2 -8821.808} C_VEL
LIN {X 0,Y 445.673,Z 671.244,A -85,B 0,C 180,E1 -8823.617,E2 -8823.617} C_VEL
LIN {X 0,Y 445.663,Z 668.766,A -85,B 0,C 180,E1 -8825.43,E2 -8825.43} C_VEL
LIN {X 0,Y 445.871,Z 665.359,A -85,B 0,C 180,E1 -8827.245,E2 -8827.245} C_VEL
LIN {X 0,Y 446.121,Z 659.554,A -85,B 0,C 180,E1 -8829.522,E2 -8829.522} C_VEL
LIN {X 0,Y 446.491,Z 653.56,A -85,B 0,C 180,E1 -8831.348,E2 -8831.348} C_VEL
LIN {X 0,Y 447.009,Z 646.296,A -85,B 0,C 180,E1 -8833.178,E2 -8833.178} C_VEL
LIN {X 0,Y 447.727,Z 637.548,A -85,B 0,C 180,E1 -8835.011,E2 -8835.011} C_VEL
LIN {X 0,Y 448.653,Z 627.742,A -85,B 0,C 180,E1 -8836.742,E2 -8836.742} C_VEL
LIN {X 0,Y 449.676,Z 616.216,A -85,B 0,C 180,E1 -8838.451,E2 -8838.451} C_VEL
LIN {X 0,Y 450.732,Z 605.286,A -85,B 0,C 180,E1 -8839.825,E2 -8839.825} C_VEL
LIN {X 0,Y 451.958,Z 591.885,A -85,B 0,C 180,E1 -8841.268,E2 -8841.268} C_VEL
LIN {X 0,Y 453.143,Z 578.883,A -85,B 0,C 180,E1 -8842.453,E2 -8842.453} C_VEL
LIN {X 0,Y 454.285,Z 565.521,A -85,B 0,C 180,E1 -8843.476,E2 -8843.476} C_VEL
LIN {X 0,Y 455.331,Z 550.582,A -85,B 0,C 180,E1 -8844.434,E2 -8844.434} C_VEL
LIN {X 0,Y 456.374,Z 534.443,A -85,B 0,C 180,E1 -8845.264,E2 -8845.264} C_VEL
LIN {X 0,Y 456.591,Z 527.686,A -85,B 0,C 180,E1 -8845.567,E2 -8845.567} C_VEL
